FUNCTION "G7_STD_3" : VOID	// FC 72
AUTHOR : SIMATIC
FAMILY : S7GRAPH
NAME : SFMULTI
VERSION : 2.0
BEGIN
// (block stored without names or comments; labels and parameter names are numbered)
NETWORK
TITLE =
// (network holds code this reader does not know; not shown)
NETWORK
TITLE =
      L     DID [AR1,P#80.0];
      LAR2;
      L     DID [AR2,P#14.0];
      T     LD 30;
      L     DID [AR2,P#18.0];
      T     LD 40;
      L     DID [AR1,P#48.0];
      AD    DW#16#7FFFF;
      LAR2;
      AN    L 30.7;
      JC    M007;
      A     DIX [AR2,P#0.0];
      FP    DIX [AR1,P#7.4];
      S     DIX [AR1,P#11.4];
      +AR2  P#0.1;
M007: AN    L 30.6;
      JC    M008;
      A     DIX [AR2,P#0.0];
      FP    DIX [AR1,P#7.5];
      S     DIX [AR1,P#11.5];
      +AR2  P#0.1;
M008: AN    L 30.5;
      JC    M009;
      A     DIX [AR2,P#0.0];
      FP    DIX [AR1,P#9.3];
      S     DIX [AR1,P#13.3];
      +AR2  P#0.1;
M009: AN    L 30.4;
      JC    M010;
      A     DIX [AR2,P#0.0];
      FP    DIX [AR1,P#9.2];
      S     DIX [AR1,P#13.2];
      +AR2  P#0.1;
M010: AN    L 30.3;
      JC    M011;
      A     DIX [AR2,P#0.0];
      FP    DIX [AR1,P#6.4];
      S     DIX [AR1,P#10.4];
      +AR2  P#0.1;
M011: AN    L 30.2;
      JC    M012;
      A     DIX [AR2,P#0.0];
      FP    DIX [AR1,P#6.5];
      S     DIX [AR1,P#10.5];
      +AR2  P#0.1;
M012: AN    L 30.1;
      JC    M013;
      A     DIX [AR2,P#0.0];
      FP    DIX [AR1,P#7.6];
      X     DIX [AR1,P#11.6];
      =     DIX [AR1,P#11.6];
      +AR2  P#0.1;
M013: AN    L 30.0;
      JC    M014;
      A     DIX [AR2,P#0.0];
      FP    DIX [AR1,P#7.7];
      X     DIX [AR1,P#11.7];
      =     DIX [AR1,P#11.7];
      +AR2  P#0.1;
M014: AN    L 31.7;
      JC    M015;
      A     DIX [AR2,P#0.0];
      FP    DIX [AR1,P#8.0];
      X     DIX [AR1,P#12.0];
      =     DIX [AR1,P#12.0];
      +AR2  P#0.1;
M015: AN    L 31.6;
      JC    M016;
      A     DIX [AR2,P#0.0];
      FP    DIX [AR1,P#7.0];
      X     DIX [AR1,P#11.0];
      =     DIX [AR1,P#11.0];
      +AR2  P#0.1;
M016: AN    L 31.5;
      JC    M017;
      A     DIX [AR2,P#0.0];
      FP    DIX [AR1,P#7.1];
      X     DIX [AR1,P#11.1];
      =     DIX [AR1,P#11.1];
      +AR2  P#0.1;
M017: AN    L 31.4;
      JC    M018;
      A     DIX [AR2,P#0.0];
      FP    DIX [AR1,P#7.2];
      X     DIX [AR1,P#11.2];
      =     DIX [AR1,P#11.2];
      +AR2  P#0.1;
M018: AN    L 31.3;
      JC    M019;
      A     DIX [AR2,P#0.0];
      FP    DIX [AR1,P#7.3];
      X     DIX [AR1,P#11.3];
      =     DIX [AR1,P#11.3];
      +AR2  P#0.1;
M019: AN    L 31.2;
      JC    M020;
      A     DIX [AR2,P#0.0];
      FP    DIX [AR1,P#8.1];
      S     DIX [AR1,P#12.1];
      R     DIX [AR1,P#12.2];
      R     DIX [AR1,P#12.3];
      R     DIX [AR1,P#12.4];
      R     DIX [AR1,P#12.5];
      +AR2  P#0.1;
M020: AN    L 31.1;
      JC    M021;
      A     DIX [AR2,P#0.0];
      FP    DIX [AR1,P#8.2];
      R     DIX [AR1,P#12.1];
      S     DIX [AR1,P#12.2];
      R     DIX [AR1,P#12.3];
      R     DIX [AR1,P#12.4];
      R     DIX [AR1,P#12.5];
      +AR2  P#0.1;
M021: AN    L 31.0;
      JC    M022;
      A     DIX [AR2,P#0.0];
      FP    DIX [AR1,P#8.3];
      R     DIX [AR1,P#12.1];
      R     DIX [AR1,P#12.2];
      S     DIX [AR1,P#12.3];
      R     DIX [AR1,P#12.4];
      R     DIX [AR1,P#12.5];
      +AR2  P#0.1;
M022: AN    L 32.7;
      JC    M023;
      A     DIX [AR2,P#0.0];
      FP    DIX [AR1,P#8.4];
      S     DIX [AR1,P#12.4];
      +AR2  P#0.1;
M023: AN    L 32.6;
      JC    M024;
      A     DIX [AR2,P#0.0];
      FP    DIX [AR1,P#8.5];
      S     DIX [AR1,P#12.5];
      +AR2  P#0.1;
M024: AN    L 32.5;
      JC    M025;
      A     DIX [AR2,P#0.0];
      FP    DIX [AR1,P#6.0];
      =     L 29.1;
      S     DIX [AR1,P#10.0];
      R     DIX [AR1,P#10.2];
      R     DIX [AR1,P#10.3];
      R     DIX [AR1,P#10.1];
      +AR2  P#0.1;
      R     DIX [AR1,P#12.4];
      R     DIX [AR1,P#12.5];
      R     DIX [AR1,P#10.6];
      R     DIX [AR1,P#10.7];
      AN    L 31.2;
      AN    L 31.1;
      AN    L 31.0;
      A     L 29.1;
      S     DIX [AR1,P#12.1];
      R     DIX [AR1,P#12.2];
      R     DIX [AR1,P#12.3];
M025: AN    L 32.4;
      JC    M026;
      A     DIX [AR2,P#0.0];
      FP    DIX [AR1,P#6.2];
      =     L 29.1;
      R     DIX [AR1,P#10.0];
      S     DIX [AR1,P#10.2];
      R     DIX [AR1,P#10.3];
      R     DIX [AR1,P#10.1];
      +AR2  P#0.1;
      R     DIX [AR1,P#12.4];
      R     DIX [AR1,P#12.5];
      R     DIX [AR1,P#10.6];
      R     DIX [AR1,P#10.7];
      AN    L 31.2;
      AN    L 31.1;
      AN    L 31.0;
      A     L 29.1;
      S     DIX [AR1,P#12.1];
      R     DIX [AR1,P#12.2];
      R     DIX [AR1,P#12.3];
M026: AN    L 32.3;
      JC    M027;
      A     DIX [AR2,P#0.0];
      FP    DIX [AR1,P#6.3];
      =     L 29.1;
      R     DIX [AR1,P#10.0];
      R     DIX [AR1,P#10.2];
      S     DIX [AR1,P#10.3];
      R     DIX [AR1,P#10.1];
      +AR2  P#0.1;
      R     DIX [AR1,P#12.4];
      R     DIX [AR1,P#12.5];
      R     DIX [AR1,P#10.6];
      R     DIX [AR1,P#10.7];
      AN    L 31.2;
      AN    L 31.1;
      AN    L 31.0;
      A     L 29.1;
      S     DIX [AR1,P#12.1];
      R     DIX [AR1,P#12.2];
      R     DIX [AR1,P#12.3];
M027: AN    L 32.2;
      JC    M028;
      A     DIX [AR2,P#0.0];
      FP    DIX [AR1,P#6.1];
      =     L 29.1;
      R     DIX [AR1,P#10.0];
      R     DIX [AR1,P#10.2];
      R     DIX [AR1,P#10.3];
      S     DIX [AR1,P#10.1];
      +AR2  P#0.1;
      R     DIX [AR1,P#12.4];
      R     DIX [AR1,P#12.5];
      R     DIX [AR1,P#10.6];
      R     DIX [AR1,P#10.7];
      AN    L 31.2;
      AN    L 31.1;
      AN    L 31.0;
      A     L 29.1;
      R     DIX [AR1,P#12.1];
      R     DIX [AR1,P#12.2];
      S     DIX [AR1,P#12.3];
M028: AN    L 32.1;
      JC    M031;
      +AR2  P#1.7;
      TAR2;
      SRD   4;
      SLD   4;
      LAR2;
      AN    L 32.0;
      JC    M029;
      L     DIW [AR2,P#0.0];
      T     DIW [AR1,P#2.0];
      JU    M030;
M029: L     DIW [AR1,P#2.0];
      L     DIW [AR2,P#0.0];
      T     DIW [AR1,P#2.0];
      <>I;
      S     DIX [AR1,P#12.6];
M030: +AR2  P#2.0;
M031: AN    L 32.0;
      JC    M032;
      A     DIX [AR2,P#0.0];
      FP    DIX [AR1,P#8.6];
      S     DIX [AR1,P#12.6];
      +AR2  P#0.1;
M032: AN    L 33.7;
      JC    M033;
      A     DIX [AR2,P#0.0];
      FP    DIX [AR1,P#8.7];
      S     DIX [AR1,P#12.7];
      +AR2  P#0.1;
M033: AN    L 33.6;
      JC    M034;
      A     DIX [AR2,P#0.0];
      FP    DIX [AR1,P#9.0];
      S     DIX [AR1,P#13.0];
      +AR2  P#0.1;
M034: AN    L 33.5;
      JC    M035;
      A     DIX [AR2,P#0.0];
      FP    DIX [AR1,P#6.6];
      S     DIX [AR1,P#10.6];
      +AR2  P#0.1;
M035: AN    L 33.4;
      JC    M036;
      A     DIX [AR2,P#0.0];
      FP    DIX [AR1,P#6.7];
      S     DIX [AR1,P#10.7];
      +AR2  P#0.1;
M036: AN    L 33.3;
      JC    M037;
      A     DIX [AR2,P#0.0];
      FP    DIX [AR1,P#9.1];
      S     DIX [AR1,P#13.1];
M037: NOP   0;
NETWORK
TITLE =
      BLD   7;
      UC    "TIME_TCK";
      {     P#L 8.0 };
      BLD   8;
      L     LD 8;
      T     DID [AR1,P#22.0];
      A     DIX [AR1,P#11.7];
      JC    M038;
      L     DID [AR1,P#18.0];
      -D;
      T     DID [AR1,P#14.0];
      AD    DW#16#FFFFF000;
      JZ    M039;
M038: L     B#16#0;
      T     DID [AR1,P#14.0];
M039: L     DID [AR1,P#22.0];
      T     DID [AR1,P#18.0];
NETWORK
TITLE =
      L     DID [AR1,P#48.0];
      LAR2;
      L     DIW [AR1,P#52.0];
      T     LW 12;
      SET;
      S     DIX [AR1,P#27.5];
      AN    DIX [AR1,P#13.6];
      JC    M040;
      A     DIX [AR1,P#10.1];
      =     DIX [AR1,P#13.4];
M040: LAR1  LD 0;
      L     B#16#1;
      T     DIB [AR1,P#30.0];
      UC    FB [LW 12];
NETWORK
TITLE =
      LAR1  LD 4;
      L     DID [AR1,P#14.0];
      T     LW 22;
      CLR;
      LAR1  LD 0;
      L     DID [AR1,P#4.0];
      T     LD 8;
      LAR1;
      L     DIB [AR1,P#0.0];
      JU    M045;
M041: T     LB 16;
      +AR1  P#1.0;
      L     DIB [AR1,P#0.0];
      SLW   7;
      LAR2  LD 0;
      +AR2;
      +AR2;
      L     DID [AR2,P#4.0];
      L     LW 22;
      +D;
      <=D;
      JC    M042;
      L     DW#16#7FFFFFFF;
M042: T     DID [AR2,P#4.0];
      O     DIX [AR2,P#1.1];
      O     DIX [AR2,P#1.2];
      JC    M044;
      L     DID [AR2,P#8.0];
      L     LW 22;
      +D;
      <=D;
      JC    M043;
      L     DW#16#7FFFFFFF;
M043: T     DID [AR2,P#8.0];
M044: L     LB 16;
M045: LOOP  M041;
NETWORK
TITLE =
      LAR1  LD 4;
      L     DID [AR1,P#40.0];
      LAR1;
      SET;
      R     L 29.0;
      JU    M285;
M046: LAR1  LD 8;
      SET;
      S     L 29.0;
      JU    M285;
M047: LAR1  LD 4;
      L     DID [AR1,P#44.0];
      LAR2;
      L     B#16#1;
      T     DIB [AR2,P#0.0];
      L     DID [AR1,P#40.0];
      LAR2;
      L     B#16#1;
      T     DIB [AR2,P#0.0];
      L     DID [AR1,P#36.0];
      LAR2;
      L     B#16#1;
      T     DIB [AR2,P#0.0];
      LAR1  LD 8;
      L     B#16#0;
      JU    M251;
M048: NOP   0;
NETWORK
TITLE =
      LAR1  LD 4;
      AN    DIX [AR1,P#11.4];
      JC    M050;
      R     DIX [AR1,P#11.4];
      R     DIX [AR1,P#11.5];
      LAR1  LD 8;
      L     B#16#0;
      JU    M261;
M049: JU    M080;
M050: NOP   0;
NETWORK
TITLE =
      LAR1  LD 4;
      AN    DIX [AR1,P#11.5];
      JC    M056;
      R     DIX [AR1,P#11.5];
      R     DIX [AR1,P#26.4];
      R     DIX [AR1,P#26.5];
      R     DIX [AR1,P#26.6];
      R     DIX [AR1,P#26.7];
      R     DIX [AR1,P#27.0];
      R     DIX [AR1,P#26.3];
      LAR1  LD 8;
      L     B#16#1;
      JU    M261;
M051: LAR1  LD 0;
      L     DIW [AR1,P#28.0];
      SLD   3;
      LAR1;
      L     B#16#0;
      JU    M256;
M052: LAR1  LD 4;
      L     DID [AR1,P#40.0];
      LAR1;
      L     B#16#4;
      JU    M270;
M053: LAR1  LD 4;
      L     DID [AR1,P#36.0];
      T     LD 8;
      LAR1;
      L     B#16#3;
      JU    M270;
M054: LAR1  LD 8;
      L     B#16#1;
      JU    M251;
M055: JU    M080;
M056: NOP   0;
NETWORK
TITLE =
      LAR1  LD 4;
      AN    DIX [AR1,P#13.3];
      AN    DIX [AR1,P#13.2];
      JC    M060;
      A     DIX [AR1,P#13.3];
      R     DIX [AR1,P#26.1];
      R     DIX [AR1,P#26.2];
      R     DIX [AR1,P#26.0];
      R     DIX [AR1,P#26.4];
      R     DIX [AR1,P#26.5];
      R     DIX [AR1,P#26.6];
      R     DIX [AR1,P#26.7];
      R     DIX [AR1,P#27.0];
      R     DIX [AR1,P#26.3];
      LAR2  LD 0;
      L     DIW [AR2,P#18.0];
      SLD   3;
      T     LD 24;
      L     DIB [LD 24];
      JU    M059;
M057: T     LB 17;
      L     LD 24;
      +     L#8;
      T     LD 24;
      L     DIB [LD 24];
      SLW   7;
      LAR2  LD 0;
      +AR2;
      +AR2;
      A     DIX [AR1,P#13.2];
      S     DIX [AR2,P#0.3];
      AN    DIX [AR1,P#13.3];
      JC    M058;
      S     DIX [AR2,P#0.4];
      R     DIX [AR2,P#1.2];
      L     B#16#0;
      T     DID [AR2,P#8.0];
M058: L     LB 17;
M059: LOOP  M057;
      R     DIX [AR1,P#13.2];
M060: R     DIX [AR1,P#13.3];
NETWORK
TITLE =
      AN    DIX [AR1,P#10.4];
      AN    DIX [AR1,P#10.5];
      JC    M061;
      L     B#16#0;
      L     DIB [AR1,P#4.0];
      ==I;
      JC    M061;
      SLW   7;
      LAR2  LD 0;
      +AR2;
      +AR2;
      A     DIX [AR1,P#10.5];
      A(;
      O     DIX [AR2,P#1.1];
      O     DIX [AR2,P#1.2];
      );
      S     DIX [AR2,P#0.3];
      A     DIX [AR1,P#10.4];
      A(;
      O     DIX [AR2,P#1.1];
      O     DIX [AR2,P#1.2];
      );
      JCN   M061;
      S     DIX [AR2,P#0.4];
      R     DIX [AR2,P#1.2];
      L     B#16#0;
      T     DID [AR2,P#8.0];
M061: R     DIX [AR1,P#10.5];
      R     DIX [AR1,P#10.4];
NETWORK
TITLE =
      AN    DIX [AR1,P#12.4];
      JC    M064;
      L     B#16#0;
      L     DIB [AR1,P#4.0];
      ==I;
      JC    M064;
      L     B#16#2;
      L     DIB [AR1,P#4.0];
      >I;
      JC    M062;
      DEC   1;
      JU    M063;
M062: L     DID [AR1,P#80.0];
      LAR2;
      L     DIB [AR2,P#12.0];
M063: T     DIB [AR1,P#4.0];
      A     DIX [AR1,P#12.3];
      JC    M064;
      SLW   7;
      LAR2  LD 0;
      +AR2;
      +AR2;
      A     DIX [AR1,P#12.1];
      A     DIX [AR2,P#1.0];
      O;
      A     DIX [AR1,P#12.2];
      A(;
      O     DIX [AR2,P#1.1];
      O     DIX [AR2,P#1.2];
      );
M064: R     DIX [AR1,P#12.4];
NETWORK
TITLE =
      AN    DIX [AR1,P#12.5];
      JC    M066;
      L     B#16#0;
      L     DIB [AR1,P#4.0];
      ==I;
      JC    M066;
      L     DID [AR1,P#80.0];
      LAR2;
      L     DIB [AR2,P#12.0];
      L     DIB [AR1,P#4.0];
      INC   1;
      >=I;
      JC    M065;
      L     B#16#1;
M065: T     DIB [AR1,P#4.0];
      A     DIX [AR1,P#12.3];
      JC    M066;
      SLW   7;
      LAR2  LD 0;
      +AR2;
      +AR2;
      A     DIX [AR1,P#12.1];
      A     DIX [AR2,P#1.0];
      O;
      A     DIX [AR1,P#12.2];
      A(;
      O     DIX [AR2,P#1.1];
      O     DIX [AR2,P#1.2];
      );
M066: R     DIX [AR1,P#12.5];
NETWORK
TITLE =
      ON    DIX [AR1,P#10.1];
      ON    DIX [AR1,P#12.6];
      JC    M068;
      L     DIW [AR1,P#2.0];
      L     B#16#2;
      JU    M266;
M067: TAK;
      L     B#16#0;
      ==I;
      JC    M068;
      TAK;
      T     DIB [AR1,P#4.0];
M068: R     DIX [AR1,P#12.6];
NETWORK
TITLE =
      AN    DIX [AR1,P#10.1];
      R     DIX [AR1,P#12.7];
      AN    DIX [AR1,P#12.7];
      JC    M070;
      R     DIX [AR1,P#12.7];
      L     DIW [AR1,P#0.0];
      L     B#16#0;
      JU    M266;
M069: <>I;
      R     L 29.0;
      TAK;
      JC    M288;
M070: LAR1  LD 4;
      L     DID [AR1,P#68.0];
      T     LD 8;
      LAR1;
      LAR2  LD 0;
      L     DIB [AR2,P#26.0];
      SLW   3;
      +AR1;
      L     B#16#1;
      JU    M256;
M071: NOP   0;
NETWORK
TITLE =
      LAR1  LD 4;
      AN    DIX [AR1,P#10.1];
      R     DIX [AR1,P#13.0];
      AN    DIX [AR1,P#13.0];
      JC    M073;
      R     DIX [AR1,P#13.0];
      LAR2  LD 0;
      L     DID [AR2,P#4.0];
      LAR2;
      L     DIB [AR2,P#0.0];
      L     B#16#1;
      ==I;
      S     DIX [AR1,P#26.5];
      JC    M073;
      L     DIW [AR1,P#0.0];
      L     B#16#1;
      JU    M266;
M072: TAK;
      L     B#16#0;
      <>I;
      S     L 29.0;
      TAK;
      JC    M288;
M073: LAR1  LD 8;
      L     B#16#2;
      JU    M261;
M074: NOP   0;
NETWORK
TITLE =
      LAR1  LD 4;
      AN    DIX [AR1,P#10.6];
      JC    M077;
      L     B#16#0;
      L     DIB [AR1,P#5.0];
      ==I;
      JC    M077;
      L     B#16#2;
      L     DIB [AR1,P#5.0];
      >I;
      JC    M075;
      DEC   1;
      JU    M076;
M075: L     DID [AR1,P#80.0];
      LAR2;
      L     DIB [AR2,P#9.0];
M076: T     DIB [AR1,P#5.0];
      LAR2  LD 0;
      L     DIW [AR2,P#12.0];
      SLD   3;
      LAR2;
      TAK;
      SLW   7;
      +AR2;
      O(;
      O     DIX [AR1,P#10.0];
      O     DIX [AR1,P#10.3];
      A     DIX [AR2,P#0.0];
      );
      O(;
      O     DIX [AR1,P#10.1];
      O     DIX [AR1,P#10.2];
      A     DIX [AR2,P#0.1];
      );
M077: R     DIX [AR1,P#10.6];
NETWORK
TITLE =
      AN    DIX [AR1,P#10.7];
      JC    M079;
      L     B#16#0;
      L     DIB [AR1,P#5.0];
      ==I;
      JC    M079;
      L     DID [AR1,P#80.0];
      LAR2;
      L     DIB [AR2,P#9.0];
      L     DIB [AR1,P#5.0];
      INC   1;
      >=I;
      JC    M078;
      L     B#16#1;
M078: T     DIB [AR1,P#5.0];
      LAR2  LD 0;
      L     DIW [AR2,P#12.0];
      SLD   3;
      LAR2;
      TAK;
      SLW   7;
      +AR2;
      O(;
      O     DIX [AR1,P#10.0];
      O     DIX [AR1,P#10.3];
      A     DIX [AR2,P#0.0];
      );
      O(;
      O     DIX [AR1,P#10.1];
      O     DIX [AR1,P#10.2];
      A     DIX [AR2,P#0.1];
      );
M079: R     DIX [AR1,P#10.7];
NETWORK
TITLE =
M080: LAR1  LD 4;
      L     DID [AR1,P#68.0];
      LAR1;
      L     B#16#1;
      T     DIB [AR1,P#0.0];
      LAR2  LD 0;
      L     DIB [AR2,P#26.0];
      SLW   3;
      +AR1;
      TAK;
      T     DIB [AR1,P#0.0];
NETWORK
TITLE =
M081: SET;
      LAR1  LD 0;
      L     DIW [AR1,P#12.0];
      SLD   3;
      T     LD 8;
      L     DIW [AR1,P#14.0];
      SLD   3;
      LAR1;
      L     DIB [AR1,P#0.0];
      JU    M083;
M082: +AR1  P#1.0;
      L     DIB [AR1,P#0.0];
      SLW   7;
      LAR2  LD 8;
      +AR2;
      R     DIX [AR2,P#0.0];
      R     DIX [AR2,P#0.1];
      R     DIX [AR2,P#0.2];
      TAK;
M083: LOOP  M082;
      LAR1  LD 0;
      L     DIW [AR1,P#14.0];
      SLD   3;
      LAR2;
      L     B#16#1;
      T     DIB [AR2,P#0.0];
      L     DIB [AR1,P#25.0];
      SLW   3;
      +AR2;
      L     B#16#1;
      T     DIB [AR2,P#0.0];
      TAK;
      +AR2;
      L     B#16#1;
      T     DIB [AR2,P#0.0];
NETWORK
TITLE =
      LAR1  LD 4;
      L     DID [AR1,P#44.0];
      T     LD 8;
      L     DID [AR1,P#80.0];
      LAR2;
      L     DIB [AR2,P#6.0];
      T     LW 22;
      LAR2  LD 0;
      L     DIW [AR2,P#20.0];
      L     DIB [AR2,P#2.0];
      SLW   1;
      +D;
      SLD   3;
      T     LD 24;
      L     DIW [AR2,P#22.0];
      SLD   3;
      T     LD 4;
      L     DIB [LD 8];
      JU    M093;
M084: T     LB 17;
      L     LD 8;
      +     L#8;
      T     LD 8;
      L     DIB [LD 8];
      T     LB 14;
M085: SLW   7;
      LAR1  AR2;
      +AR1;
      +AR1;
      ON    DIX [AR1,P#24.0];
      O     DIX [AR1,P#0.5];
      JC    M092;
      LAR1  LD 4;
      SRW   4;
      +AR1;
      L     LB 14;
      L     DIB [AR1,P#0.0];
      <>I;
      JC    M085;
      LAR1  LD 4;
      SLW   3;
      +AR1;
      L     DIB [AR2,P#3.0];
      SLW   3;
      +AR1;
      +AR1;
      +AR1;
      L     DIB [AR1,P#0.0];
      T     LB 16;
      L     DIW [AR2,P#12.0];
      SLD   3;
      LAR1;
      TAK;
      SLW   7;
      +AR1;
      A     DIX [AR1,P#0.0];
      JC    M092;
      SRW   7;
M086: T     LB 15;
      L     DIW [AR2,P#20.0];
      SLD   3;
      LAR1;
      TAK;
      SLW   3;
      +AR1;
      L     DIB [AR1,P#0.0];
      L     DIB [AR2,P#2.0];
      SLW   5;
      +AR1;
      TAK;
      L     DIB [AR1,P#0.0];
      <>I;
      JC    M087;
      SLW   7;
      LAR1  AR2;
      +AR1;
      +AR1;
      A     DIX [AR1,P#24.0];
      JC    M092;
      JU    M089;
M087: T     LB 14;
M088: SLW   7;
      LAR1  AR2;
      +AR1;
      +AR1;
      A     DIX [AR1,P#24.0];
      JC    M092;
      L     DIB [AR2,P#3.0];
      SLW   3;
      LAR1  LD 4;
      +AR1;
      TAK;
      SRW   4;
      +AR1;
      L     LB 14;
      L     DIB [AR1,P#0.0];
      <>I;
      JC    M088;
M089: LAR1  LD 24;
      L     LB 15;
      SLW   3;
      +AR1;
      L     LB 16;
      L     DIB [AR1,P#0.0];
      <>I;
      JC    M086;
M090: T     LB 15;
      L     DIW [AR2,P#14.0];
      SLD   3;
      LAR1;
      L     LW 22;
      L     DIB [AR1,P#0.0];
      >=I;
      JC    M091;
      L     DID [AR2,P#8.0];
      LAR1;
      S     DIX [AR1,P#26.7];
      JU    M094;
M091: INC   1;
      T     DIB [AR1,P#0.0];
      DEC   1;
      SLW   3;
      +AR1;
      L     LB 15;
      T     DIB [AR1,P#0.0];
      L     DIW [AR2,P#12.0];
      SLD   3;
      LAR1;
      TAK;
      SLW   7;
      +AR1;
      S     DIX [AR1,P#0.0];
      LAR1  LD 24;
      SRW   4;
      +AR1;
      L     LB 16;
      L     DIB [AR1,P#0.0];
      <>I;
      JC    M090;
M092: L     LB 17;
M093: LOOP  M084;
M094: L     DID [AR2,P#8.0];
      T     LD 4;
NETWORK
TITLE =
      LAR1  LD 4;
      CLR;
      A     DIX [AR1,P#13.5];
      =     L 29.7;
      O     DIX [AR1,P#10.6];
      O     DIX [AR1,P#10.7];
      A     L 41.6;
      R     DIX [AR1,P#13.1];
      L     DIW [AR2,P#14.0];
      SLD   3;
      T     LD 8;
      LAR1;
      L     DIB [AR2,P#25.0];
      SLW   3;
      T     LW 22;
      +D;
      T     LD 24;
      L     DIB [AR1,P#0.0];
      T     LB 16;
      SLW   3;
      +AR1;
      L     B#16#0;
      T     DIB [AR1,P#0.0];
      T     LB 15;
      AN    L 29.7;
      JC    M095;
      LAR1  LD 4;
      L     DID [AR1,P#80.0];
      LAR1;
      L     DIB [AR1,P#9.0];
      INC   1;
      T     LB 16;
M095: L     LB 16;
      JU    M101;
M096: T     LB 16;
      LAR1  LD 4;
      L     B#16#0;
      T     DID [AR1,P#72.0];
      L     DID [AR1,P#48.0];
      LAR2;
      A     L 29.7;
      JC    M097;
      L     LD 8;
      +     L#8;
      T     LD 8;
      L     DIB [LD 8];
      JU    M098;
M097: L     LB 15;
      INC   1;
M098: T     LB 15;
      LAR1  LD 0;
      T     DIB [AR1,P#31.0];
      L     B#16#2;
      T     DIB [AR1,P#30.0];
      UC    FB [LW 12];
      LAR1  LD 0;
      L     DIW [AR1,P#12.0];
      SLD   3;
      LAR1;
      L     LB 15;
      SLW   7;
      +AR1;
      =     DIX [AR1,P#0.1];
      LAR2  LD 4;
      AN    DIX [AR1,P#0.0];
      JC    M099;
      O(;
      SRW   7;
      L     DIB [AR2,P#5.0];
      ==I;
      A     L 41.6;
      A     DIX [AR2,P#10.3];
      A     DIX [AR2,P#13.1];
      );
      O(;
      AN    L 41.6;
      A     DIX [AR2,P#10.3];
      A     DIX [AR2,P#13.1];
      );
      R     DIX [AR2,P#13.1];
      S     DIX [AR1,P#0.1];
      L     DID [AR1,P#4.0];
      T     DID [AR1,P#8.0];
M099: L     DID [AR2,P#72.0];
      T     DID [AR1,P#4.0];
      ON    DIX [AR1,P#0.0];
      ON    DIX [AR1,P#0.1];
      JC    M100;
      LAR1  LD 24;
      L     DIB [AR1,P#0.0];
      INC   1;
      T     DIB [AR1,P#0.0];
      DEC   1;
      SLW   3;
      +AR1;
      L     LB 15;
      T     DIB [AR1,P#0.0];
M100: L     LB 16;
M101: LOOP  M096;
NETWORK
TITLE =
// (network holds code this reader does not know; not shown)
NETWORK
TITLE =
// (network holds code this reader does not know; not shown)
NETWORK
TITLE =
      LAR1  LD 0;
      L     DIB [AR1,P#2.0];
      SLW   3;
      L     LD 24;
      +D;
      T     LD 24;
      L     DID [AR1,P#8.0];
      LAR1;
      L     DID [AR1,P#36.0];
      T     LD 4;
      LAR2  LD 8;
      L     DIB [AR2,P#0.0];
      JU    M117;
M113: T     LB 17;
      +AR2  P#1.0;
      LAR1  LD 24;
      L     DIB [AR2,P#0.0];
      T     LB 15;
      SLW   3;
      +AR1;
      L     B#16#0;
      L     DIB [AR1,P#0.0];
      ==I;
      JC    M116;
      T     LB 14;
M114: T     LB 16;
      SLW   7;
      LAR1  LD 0;
      +AR1;
      +AR1;
      O     DIX [AR1,P#0.0];
      O     DIX [AR1,P#1.0];
      JC    M115;
      S     DIX [AR1,P#0.0];
      S     DIX [AR1,P#1.0];
      LAR1  LD 4;
      L     DIB [AR1,P#0.0];
      INC   1;
      T     DIB [AR1,P#0.0];
      DEC   1;
      SLW   3;
      +AR1;
      L     LB 16;
      T     DIB [AR1,P#0.0];
      LAR1  LD 0;
      L     DIW [AR1,P#20.0];
      SLD   3;
      LAR1;
      L     LB 15;
      SLW   3;
      +AR1;
      L     DIB [AR1,P#0.0];
      L     B#16#0;
      <>I;
      JC    M116;
M115: LAR1  LD 0;
      L     DIW [AR1,P#22.0];
      L     DIB [AR1,P#3.0];
      +D;
      SLD   3;
      LAR1;
      L     LB 16;
      SLW   3;
      +AR1;
      L     LB 14;
      L     DIB [AR1,P#0.0];
      <>I;
      JC    M114;
M116: L     LB 17;
M117: LOOP  M113;
NETWORK
TITLE =
      LAR1  LD 4;
      LAR2  LD 0;
      L     DID [AR2,P#8.0];
      T     LD 4;
      L     B#16#2;
      JU    M251;
M118: NOP   0;
NETWORK
TITLE =
      LAR1  LD 8;
      LAR2  LD 4;
      L     B#16#1;
      L     DIB [AR1,P#0.0];
      <I;
      A     DIX [AR2,P#11.3];
      JC    M081;
NETWORK
TITLE =
      L     DID [AR2,P#44.0];
      LAR1;
      L     DIB [AR1,P#0.0];
      JU    M120;
M119: +AR1  P#1.0;
      L     DIB [AR1,P#0.0];
      SLW   7;
      LAR2  LD 0;
      +AR2;
      +AR2;
      R     DIX [AR2,P#24.0];
      TAK;
M120: LOOP  M119;
NETWORK
TITLE =
      LAR1  LD 4;
      L     DID [AR1,P#80.0];
      LAR2;
      AN    DIX [AR2,P#34.7];
      JC    M129;
      L     DIW [AR2,P#32.0];
      T     LW 18;
      L     B#16#2;
      -D;
      SLD   3;
      LAR2;
      L     DIW [AR2,P#0.0];
      T     LW 20;
      L     LW 18;
      LAR2  LD 0;
      L     DIB [AR2,P#3.0];
      INC   2;
      -D;
      SLD   3;
      T     LD 8;
      L     DIB [LD 8];
      T     LW 18;
      L     DID [AR1,P#36.0];
      T     LD 24;
      L     DIB [LD 24];
      JU    M128;
M121: T     LB 17;
      L     LD 24;
      +     L#8;
      T     LD 24;
      L     DIB [LD 24];
      SLW   3;
      LAR1  LD 8;
      +AR1;
      L     DIB [AR1,P#0.0];
      T     LW 22;
      SET;
      =     L 29.6;
      LAR1  LD 0;
      L     DID [AR1,P#4.0];
      LAR2;
M122: L     DIB [AR2,P#0.0];
      JU    M126;
M123: T     LB 14;
      +AR2  P#1.0;
      L     DIB [LD 24];
      L     DIB [AR2,P#0.0];
      <>I;
      JC    M124;
      A     L 29.6;
      JC    M125;
      L     B#16#1;
      T     LB 14;
      JC    M125;
M124: T     LB 16;
      SLW   3;
      LAR1  LD 8;
      +AR1;
      L     DIB [AR1,P#0.0];
      L     LW 18;
      *D;
      L     LW 22;
      +D;
      L     LW 20;
      SLD   3;
      +D;
      LAR1;
      A     DIX [AR1,P#0.0];
      JC    M125;
      L     LB 16;
      SLW   7;
      LAR1  LD 0;
      +AR1;
      +AR1;
      O     DIX [AR1,P#0.5];
      ON    DIX [AR1,P#1.0];
      JC    M125;
      S     DIX [AR1,P#0.5];
      R     DIX [AR1,P#1.0];
      LAR1  LD 4;
      L     DID [AR1,P#40.0];
      LAR1;
      L     DIB [AR1,P#0.0];
      INC   1;
      T     DIB [AR1,P#0.0];
      DEC   1;
      SLW   3;
      +AR1;
      L     LB 16;
      T     DIB [AR1,P#0.0];
M125: L     LB 14;
M126: LOOP  M123;
      AN    L 29.6;
      JC    M127;
      R     L 29.6;
      LAR1  LD 4;
      L     DID [AR1,P#36.0];
      LAR2;
      JU    M122;
M127: L     LB 17;
M128: LOOP  M121;
M129: NOP   0;
NETWORK
TITLE =
      LAR1  LD 4;
      L     DID [AR1,P#40.0];
      LAR1;
      L     B#16#2;
      JU    M270;
M130: NOP   0;
NETWORK
TITLE =
      LAR1  LD 4;
      L     DID [AR1,P#36.0];
      T     LD 8;
      LAR1;
      L     B#16#1;
      JU    M270;
M131: NOP   0;
NETWORK
TITLE =
      LAR1  LD 8;
      L     DIB [AR1,P#0.0];
      JU    M133;
M132: T     LB 14;
      +AR1  P#1.0;
      L     DIB [AR1,P#0.0];
      SLW   7;
      LAR2  LD 0;
      +AR2;
      +AR2;
      L     B#16#0;
      T     DID [AR2,P#4.0];
      T     DID [AR2,P#8.0];
      L     LB 14;
M133: LOOP  M132;
NETWORK
TITLE =
      LAR1  LD 0;
      L     DID [AR1,P#4.0];
      T     LD 8;
      LAR2;
      LAR1  LD 4;
      L     DID [AR1,P#44.0];
      LAR1;
      L     DIB [AR2,P#0.0];
M134: L     DIB [AR2,P#0.0];
      T     DIB [AR1,P#0.0];
      +AR1  P#1.0;
      +AR2  P#1.0;
      TAK;
      LOOP  M134;
      LAR1  LD 4;
      SET;
      S     DIX [AR1,P#27.6];
      LAR1  LD 8;
      L     B#16#0;
      JU    M270;
M135: NOP   0;
NETWORK
TITLE =
      LAR1  LD 4;
      L     DID [AR1,P#80.0];
      LAR2;
      L     DIB [AR2,P#7.0];
      T     LB 14;
      L     DID [AR1,P#36.0];
      LAR1;
      L     DIB [AR1,P#0.0];
      DEC   1;
      LAR2  LD 8;
      L     DIB [AR2,P#0.0];
      DEC   1;
      +I;
      L     LB 14;
      <=I;
      JC    M137;
      LAR2  LD 4;
      S     DIX [AR2,P#26.6];
      -I;
      T     LB 14;
      L     DIB [AR1,P#0.0];
      TAK;
      -I;
      T     DIB [AR1,P#0.0];
      SLW   3;
      +AR1;
      L     LB 14;
M136: T     LB 14;
      L     DIB [AR1,P#0.0];
      SLW   7;
      LAR2  LD 0;
      +AR2;
      +AR2;
      L     B#16#0;
      T     DIW [AR2,P#0.0];
      +AR1  P#1.0;
      L     LB 14;
      LOOP  M136;
M137: NOP   0;
NETWORK
TITLE =
// (network holds code this reader does not know; not shown)
NETWORK
TITLE =
      LAR1  LD 0;
      L     DIW [AR1,P#16.0];
      L     DIB [AR1,P#26.0];
      +D;
      SLD   3;
      LAR1;
      LAR2  LD 4;
      L     DID [AR2,P#40.0];
      LAR2;
      L     DIB [AR2,P#0.0];
M170: L     DIB [AR2,P#0.0];
      T     DIB [AR1,P#0.0];
      +AR1  P#1.0;
      +AR2  P#1.0;
      TAK;
      LOOP  M170;
      LAR1  LD 4;
      L     DID [AR1,P#36.0];
      LAR1;
      LAR2  LD 0;
      L     DID [AR2,P#4.0];
      LAR2;
      L     DIB [AR2,P#0.0];
      T     LB 14;
      L     DIB [AR1,P#0.0];
      DEC   1;
      +I;
      T     DIB [AR2,P#0.0];
      L     LB 14;
      SLW   3;
      +AR2;
      L     DIB [AR1,P#0.0];
      JU    M172;
M171: +AR1  P#1.0;
      L     DIB [AR1,P#0.0];
      T     DIB [AR2,P#0.0];
      +AR2  P#1.0;
      TAK;
M172: LOOP  M171;
      LAR1  LD 4;
      SET;
      R     DIX [AR1,P#27.6];
NETWORK
TITLE =
      LAR1  LD 0;
      L     B#16#6;
      T     DIB [AR1,P#30.0];
      LAR1  LD 4;
      L     DID [AR1,P#48.0];
      LAR2;
      UC    FB [LW 12];
      LAR1  LD 4;
      SET;
      R     DIX [AR1,P#27.5];
NETWORK
TITLE =
      LAR1  LD 0;
      L     DIW [AR1,P#18.0];
      SLD   3;
      T     LD 8;
      LAR1  LD 4;
      SET;
      R     DIX [AR1,P#26.1];
      R     DIX [AR1,P#26.2];
      L     DIB [LD 8];
      JU    M174;
M173: T     LB 14;
      L     LD 8;
      +     L#8;
      T     LD 8;
      L     DIB [LD 8];
      SLW   7;
      LAR2  LD 0;
      +AR2;
      +AR2;
      A     DIX [AR2,P#1.1];
      S     DIX [AR1,P#26.1];
      A     DIX [AR2,P#1.2];
      S     DIX [AR1,P#26.2];
      L     LB 14;
M174: LOOP  M173;
      O     DIX [AR1,P#26.1];
      O     DIX [AR1,P#26.2];
      =     DIX [AR1,P#26.0];
      O     DIX [AR1,P#26.4];
      O     DIX [AR1,P#26.5];
      O     DIX [AR1,P#26.6];
      O     DIX [AR1,P#26.7];
      O     DIX [AR1,P#27.0];
      =     DIX [AR1,P#26.3];
NETWORK
TITLE =
// (network holds code this reader does not know; not shown)
NETWORK
TITLE =
      CLR;
      AN    DIX [AR1,P#26.3];
      SAVE;
      L     DID [AR1,P#48.0];
      LAR2;
      BE;
NETWORK
TITLE =
M251: T     LB 28;
      LAR2  LD 4;
      L     DID [AR2,P#44.0];
      T     LD 24;
      CLR;
      L     DIB [AR1,P#0.0];
      JU    M254;
M252: T     LB 17;
      +AR1  P#1.0;
      L     DIB [AR1,P#0.0];
      SLW   7;
      LAR2  LD 0;
      +AR2;
      +AR2;
      A     DIX [AR2,P#24.0];
      JC    M253;
      S     DIX [AR2,P#24.0];
      LAR2  LD 24;
      L     DIB [AR2,P#0.0];
      INC   1;
      T     DIB [AR2,P#0.0];
      DEC   1;
      SLW   3;
      +AR2;
      TAK;
      SRW   7;
      T     DIB [AR2,P#0.0];
M253: L     LB 17;
M254: LOOP  M252;
      L     LB 28;
      JL    M255;
      JU    M048;
      JU    M055;
      JU    M118;
M255: NOP   0;
NETWORK
TITLE =
M256: T     LB 28;
      LAR2  LD 4;
      L     DID [AR2,P#36.0];
      T     LD 24;
      CLR;
      L     DIB [AR1,P#0.0];
      JU    M259;
M257: T     LB 17;
      +AR1  P#1.0;
      L     DIB [AR1,P#0.0];
      SLW   7;
      LAR2  LD 0;
      +AR2;
      +AR2;
      O     DIX [AR2,P#0.0];
      O     DIX [AR2,P#1.0];
      JC    M258;
      S     DIX [AR2,P#0.0];
      S     DIX [AR2,P#1.0];
      LAR2  LD 24;
      L     DIB [AR2,P#0.0];
      INC   1;
      T     DIB [AR2,P#0.0];
      DEC   1;
      SLW   3;
      +AR2;
      TAK;
      SRW   7;
      T     DIB [AR2,P#0.0];
M258: L     LB 17;
M259: LOOP  M257;
      L     LB 28;
      JL    M260;
      JU    M052;
      JU    M071;
M260: NOP   0;
NETWORK
TITLE =
M261: T     LB 28;
      LAR2  LD 4;
      L     DID [AR2,P#40.0];
      T     LD 24;
      CLR;
      L     DIB [AR1,P#0.0];
      JU    M264;
M262: T     LB 17;
      +AR1  P#1.0;
      L     DIB [AR1,P#0.0];
      SLW   7;
      LAR2  LD 0;
      +AR2;
      +AR2;
      O     DIX [AR2,P#0.5];
      ON    DIX [AR2,P#1.0];
      JC    M263;
      S     DIX [AR2,P#0.5];
      R     DIX [AR2,P#1.0];
      LAR2  LD 24;
      L     DIB [AR2,P#0.0];
      INC   1;
      T     DIB [AR2,P#0.0];
      DEC   1;
      SLW   3;
      +AR2;
      TAK;
      SRW   7;
      T     DIB [AR2,P#0.0];
M263: L     LB 17;
M264: LOOP  M262;
      L     LB 28;
      JL    M265;
      JU    M049;
      JU    M051;
      JU    M074;
M265: NOP   0;
NETWORK
TITLE =
M266: T     LB 28;
      TAK;
      T     LW 20;
      L     B#16#0;
      T     LW 18;
      L     DID [AR1,P#80.0];
      LAR2;
      L     DIB [AR2,P#12.0];
      LAR2  LD 0;
M267: T     LB 17;
      L     LW 18;
      INC   1;
      T     LW 18;
      +AR2  P#32.0;
      L     LW 20;
      L     DIW [AR2,P#2.0];
      ==I;
      L     LW 18;
      JC    M268;
      L     LB 17;
      LOOP  M267;
      S     DIX [AR1,P#26.4];
M268: L     LB 28;
      JL    M269;
      JU    M069;
      JU    M072;
      JU    M067;
M269: NOP   0;
NETWORK
TITLE =
M270: T     LB 28;
      CLR;
      TAR1  LD 24;
      L     DIB [AR1,P#0.0];
      L     B#16#1;
      T     DIB [AR1,P#0.0];
      TAK;
      JU    M278;
M271: T     LB 17;
      +AR1  P#1.0;
      L     DIB [AR1,P#0.0];
      SLW   7;
      LAR2  LD 0;
      +AR2;
      +AR2;
      L     LB 28;
      JL    M272;
      JU    M273;
      JU    M275;
      JU    M274;
      JU    M275;
      JU    M274;
M272: NOP   0;
M273: A     DIX [AR2,P#0.5];
      JC    M277;
      JU    M276;
M274: A     DIX [AR2,P#0.5];
      A     DIX [AR2,P#0.0];
      R     DIX [AR2,P#0.5];
      R     DIX [AR2,P#0.0];
      JC    M277;
      JU    M276;
M275: AN    DIX [AR2,P#0.0];
      JC    M277;
M276: LAR2  LD 24;
      L     DIB [AR2,P#0.0];
      INC   1;
      T     DIB [AR2,P#0.0];
      DEC   1;
      SLW   3;
      +AR2;
      L     DIB [AR1,P#0.0];
      T     DIB [AR2,P#0.0];
M277: L     LB 17;
M278: LOOP  M271;
      L     LB 28;
      JL    M279;
      JU    M135;
      JU    M131;
      JU    M130;
      JU    M054;
      JU    M053;
M279: NOP   0;
NETWORK
TITLE =
M280: CLR;
      LAR1  LD 0;
      L     DIW [AR1,P#18.0];
      SLD   3;
      T     LD 24;
      LAR2;
      LAR1;
      L     DIB [AR1,P#0.0];
      JU    M284;
M281: T     LB 17;
      +AR1  P#1.0;
      L     LB 14;
      L     DIB [AR1,P#0.0];
      <>I;
      JC    M282;
      L     DIB [LD 24];
      DEC   1;
      T     DIB [LD 24];
      JU    M283;
M282: +AR2  P#1.0;
      T     DIB [AR2,P#0.0];
M283: L     LB 17;
M284: LOOP  M281;
      A     L 29.0;
      JC    M162;
      JU    M150;
NETWORK
TITLE =
M285: L     DIB [AR1,P#0.0];
      JU    M287;
M286: T     LB 17;
      +AR1  P#1.0;
      L     DIB [AR1,P#0.0];
      SLW   7;
      LAR2  LD 0;
      +AR2;
      +AR2;
      L     B#16#0;
      T     DIB [AR2,P#0.0];
      L     LB 17;
M287: LOOP  M286;
      CLR;
      A     L 29.0;
      JC    M047;
      JU    M046;
NETWORK
TITLE =
M288: T     LW 20;
      LAR1  LD 4;
      L     DID [AR1,P#68.0];
      LAR1;
      CLR;
      A     L 29.0;
      JC    M289;
      LAR2  LD 0;
      L     DIB [AR2,P#26.0];
      SLW   3;
      +AR1;
M289: LAR2  LD 4;
      L     DID [AR2,P#80.0];
      LAR2;
      L     DIB [AR2,P#7.0];
      L     DIB [AR1,P#0.0];
      <I;
      LAR2  LD 4;
      S     DIX [AR2,P#26.5];
      JC    M290;
      INC   1;
      T     DIB [AR1,P#0.0];
      DEC   1;
      SLW   3;
      +AR1;
      L     LW 20;
      T     DIB [AR1,P#0.0];
M290: A     L 29.0;
      JC    M073;
      JU    M070;
NETWORK
TITLE =
// (network holds code this reader does not know; not shown)
NETWORK
TITLE =
M318: L     DINO;
      L     DID [AR1,P#52.0];
      +D;
      T     DID [AR1,P#52.0];
      SRD   16;
      T     LW 12;
      BLD   7;
      UC    "TIME_TCK";
      {     P#L 8.0 };
      BLD   8;
      L     LD 8;
      T     DID [AR1,P#18.0];
      L     LD 24;
      T     DID [AR1,P#80.0];
      LAR2;
      L     DID [AR1,P#48.0];
      AD    DW#16#7FFFF;
      T     LD 8;
      L     DID [AR1,P#36.0];
      +D;
      T     DID [AR1,P#36.0];
      TAK;
      L     DID [AR1,P#40.0];
      +D;
      T     DID [AR1,P#40.0];
      TAK;
      L     DID [AR1,P#44.0];
      +D;
      T     DID [AR1,P#44.0];
      TAK;
      L     DID [AR1,P#68.0];
      +D;
      T     DID [AR1,P#68.0];
      TAK;
      L     DID [AR1,P#28.0];
      +D;
      T     DID [AR1,P#28.0];
      T     LD 0;
      LAR1;
      A     L 29.1;
      JC    M321;
      L     W#16#FB;
      L     DIW [AR2,P#30.0];
      ==I;
      JC    M320;
      L     W#16#FC;
      ==I;
      JC    M319;
      L     DW#16#40000000;
      T     DID [AR2,P#14.0];
      L     DW#16#0;
      T     DID [AR2,P#18.0];
      L     B#16#2;
      JU    M322;
M319: L     DW#16#E000F6C8;
      T     DID [AR2,P#14.0];
      L     DW#16#E000800D;
      T     DID [AR2,P#18.0];
      L     B#16#A;
      JU    M322;
M320: L     DW#16#E3E0F6C8;
      T     DID [AR2,P#14.0];
      L     DW#16#E000BE0D;
      T     DID [AR2,P#18.0];
      L     B#16#A;
      JU    M322;
M321: L     DIW [AR2,P#32.0];
M322: L     LD 8;
      SRD   3;
      +D;
      T     DIW [AR1,P#12.0];
      TAR1;
      SRD   3;
      L     DIB [AR2,P#12.0];
      T     LB 14;
      INC   1;
      SLW   5;
      +D;
      L     DIW [AR2,P#0.0];
      SLD   2;
      +D;
      L     DIW [AR2,P#2.0];
      SLD   2;
      +D;
      T     DIW [AR1,P#14.0];
      L     DIB [AR2,P#9.0];
      T     LB 15;
      INC   2;
      SRW   1;
      SLW   1;
      T     DIB [AR1,P#2.0];
      L     LB 14;
      INC   2;
      SRW   1;
      SLW   1;
      T     DIB [AR1,P#3.0];
      L     DIB [AR2,P#6.0];
      INC   3;
      SRW   1;
      SLW   1;
      T     DIB [AR1,P#25.0];
      L     DIB [AR2,P#7.0];
      INC   3;
      SRW   1;
      SLW   1;
      T     DIB [AR1,P#26.0];
      L     LB 14;
      INC   3;
      SRW   1;
      SLW   1;
      T     DIB [AR1,P#27.0];
      L     LD 4;
      T     DID [AR1,P#8.0];
      L     DIW [AR1,P#14.0];
      L     DIB [AR1,P#25.0];
      SLW   1;
      +D;
      T     DIW [AR1,P#16.0];
      L     DIB [AR1,P#26.0];
      SLW   2;
      +D;
      SLD   3;
      T     DID [AR1,P#4.0];
      SRD   3;
      L     DIB [AR1,P#26.0];
      +D;
      T     DIW [AR1,P#18.0];
      TAR2;
      SRD   3;
      L     DIB [AR1,P#3.0];
      SLW   2;
      -D;
      T     DIW [AR1,P#22.0];
      L     DIB [AR1,P#2.0];
      SLW   2;
      -D;
      L     DIB [AR1,P#2.0];
      -D;
      T     DIW [AR1,P#20.0];
      L     DIB [AR1,P#26.0];
      -D;
      T     DIW [AR1,P#28.0];
      A     L 29.1;
      JC    M323;
      L     DIW [AR2,P#32.0];
      JU    M324;
M323: L     DIW [AR2,P#28.0];
M324: L     W#16#105;
      ==I;
      JC    M325;
      TAK;
      L     W#16#107;
      <>I;
      JC    M328;
M325: L     DIW [AR1,P#12.0];
      SLD   3;
      LAR2;
      L     B#16#0;
      L     LB 14;
M326: +AR1  P#32.0;
      TAK;
      INC   1;
      T     DIB [AR1,P#3.0];
      S     DIX [AR1,P#1.6];
      TAK;
      LOOP  M326;
      L     LB 15;
M327: +AR2  P#16.0;
      TAK;
      INC   1;
      T     DIB [AR2,P#3.0];
      S     DIX [AR2,P#0.3];
      TAK;
      LOOP  M327;
      LAR1  LD 0;
      L     B#16#7;
      T     DIB [AR1,P#30.0];
      LAR1  LD 4;
      L     DID [AR1,P#48.0];
      LAR2;
      UC    FB [LW 12];
M328: LAR1  LD 4;
      SET;
      S     DIX [AR1,P#27.2];
      JU    M005;
NETWORK
TITLE =
// (network holds code this reader does not know; not shown)
END_FUNCTION

FUNCTION "TE-ANEI" : VOID	// FC 78
AUTHOR : SIMATIC
FAMILY : EA_DIS
NAME : TE_ANEI
VERSION : 3.0
BEGIN
// (block stored without names or comments; labels and parameter names are numbered)
NETWORK
TITLE =
      L     #PARAM12;
      L     31;
      AW;
      T     MB 200;
      L     #PARAM4;
      T     MW 210;
      A     M 200.0;
      JC    M003;
      L     #PARAM3;
      T     MW 202;
      L     #PARAM1;
      L     W#16#4550;
      ==I;
      JC    M001;
      L     MB 203;
      SLW   3;
      LAR1;
      L     DBW [AR1,P#0.0];
      T     MW 204;
      JU    M002;
M001: NOP   0;
      L     MB 203;
      SLW   3;
      LAR1;
      L     DBW [AR1,P#0.0];
      T     MW 204;
M002: NOP   0;
M003: NOP   0;
NETWORK
TITLE =
      L     MW 210;
      L     2;
      ==I;
      JC    M004;
      JU    M007;
M004: A     M 200.0;
      JC    M008;
      L     MW 204;
      T     MW 240;
      AN    M 240.7;
      JC    M005;
      L     MW 240;
      NEGI;
      DTR;
      L     -1.000000e+00;
      *R;
      JU    M006;
M005: L     MW 240;
      DTR;
M006: T     MD 230;
      L     MD 230;
      L     1.000000e+01;
      /R;
      T     MD 238;
      L     MD 238;
      L     #PARAM7;
      -R;
      T     MD 218;
      L     #PARAM8;
      L     #PARAM7;
      -R;
      T     MD 242;
      L     MD 218;
      L     MD 242;
      /R;
      L     1.000000e+04;
      *R;
      T     MD 214;
      JU    M009;
M007: JU    M011;
M008: JU    M010;
M009: O(;
      L     MD 230;
      L     8.501000e+03;
      >=R;
      );
      O(;
      L     MD 230;
      L     1.000000e+04;
      >=R;
      );
      =     M 240.0;
      O(;
      L     -2.001000e+03;
      L     MD 230;
      >=R;
      );
      O(;
      L     -2.430000e+03;
      L     MD 230;
      >=R;
      );
      =     M 240.1;
      O(;
      L     -2.431000e+03;
      L     MD 230;
      >=R;
      );
      O(;
      L     -3.276800e+04;
      L     MD 230;
      >=R;
      );
      =     M 240.2;
      O(;
      L     MD 230;
      L     1.000000e+04;
      >=R;
      );
      O(;
      L     MD 230;
      L     3.276700e+04;
      >=R;
      );
      =     M 240.3;
      O(;
      L     MD 230;
      L     -2.000000e+03;
      >=R;
      );
      O(;
      L     MD 230;
      L     8.500000e+03;
      >=R;
      );
      =     M 240.4;
      O(;
      A     M 240.0;
      A     M 240.3;
      A     M 240.4;
      );
      O(;
      A     M 240.1;
      A     M 240.2;
      );
      =     M 200.6;
      A     M 200.3;
      A     M 200.6;
      =     M 200.7;
      L     MD 238;
      JU    M012;
M010: R     M 200.7;
      L     #PARAM6;
      T     MD 206;
      L     #PARAM7;
      -R;
      T     MD 244;
      L     #PARAM8;
      L     #PARAM7;
      -R;
      T     MD 248;
      L     MD 244;
      L     MD 248;
      /R;
      L     1.000000e+04;
      *R;
      T     MD 214;
      L     MD 206;
      JU    M014;
M011: JU    M015;
M012: AN    M 200.7;
      ON    M 200.1;
      JC    M013;
      JU    M014;
      L     1.000000e+04;
      T     MD 214;
      L     #PARAM8;
M013: AN    M 200.7;
      ON    M 200.2;
      JC    M014;
      L     0.000000e+00;
      T     MD 214;
      L     #PARAM7;
M014: T     #PARAM10;
      L     MD 214;
      T     #PARAM11;
      L     MB 200;
      T     #PARAM12;
M015: NOP   0;
NETWORK
TITLE =
      L     MW 210;
      L     4;
      ==I;
      JC    M016;
      JU    M020;
M016: A     M 200.0;
      JC    M021;
      L     MW 204;
      T     MW 240;
      AN    M 240.7;
      JC    M018;
M017: L     MW 240;
      NEGI;
      DTR;
      L     -1.000000e+00;
      *R;
      JU    M019;
M018: L     MW 240;
      L     32760;
      >I;
      JC    M017;
      L     MW 240;
      DTR;
M019: T     MD 230;
      L     2.764800e+04;
      /R;
      L     1.000000e+04;
      *R;
      T     MD 214;
      L     #PARAM8;
      L     #PARAM7;
      -R;
      L     1.000000e+04;
      /R;
      T     MD 218;
      L     MD 214;
      L     MD 218;
      *R;
      T     MD 234;
      L     #PARAM7;
      +R;
      T     MD 238;
      JU    M022;
M020: JU    M024;
M021: JU    M023;
M022: O(;
      L     MD 230;
      L     2.764900e+04;
      >=R;
      );
      O(;
      L     MD 230;
      L     3.251100e+04;
      >=R;
      );
      =     M 240.0;
      O(;
      L     -2.764900e+04;
      L     MD 230;
      >=R;
      );
      O(;
      L     -3.251200e+04;
      L     MD 230;
      >=R;
      );
      =     M 240.1;
      O(;
      L     -3.251300e+04;
      L     MD 230;
      >=R;
      );
      O(;
      L     -3.276800e+04;
      L     MD 230;
      >=R;
      );
      =     M 240.2;
      O(;
      L     MD 230;
      L     3.251200e+04;
      >=R;
      );
      O(;
      L     MD 230;
      L     3.276700e+04;
      >=R;
      );
      =     M 240.3;
      O(;
      L     MD 230;
      L     -2.764800e+04;
      >=R;
      );
      O(;
      L     MD 230;
      L     2.764800e+04;
      >=R;
      );
      =     M 240.4;
      O(;
      A     M 240.0;
      A     M 240.3;
      A     M 240.4;
      );
      O(;
      A     M 240.1;
      A     M 240.2;
      );
      =     M 200.6;
      A     M 200.3;
      A     M 200.6;
      =     M 200.7;
      L     MD 238;
      JU    M025;
M023: R     M 200.7;
      L     #PARAM6;
      T     MD 206;
      L     #PARAM7;
      -R;
      T     MD 244;
      L     #PARAM8;
      L     #PARAM7;
      -R;
      T     MD 248;
      L     MD 244;
      L     MD 248;
      /R;
      L     1.000000e+04;
      *R;
      T     MD 214;
      L     MD 206;
      JU    M027;
M024: JU    M028;
M025: AN    M 200.7;
      ON    M 200.1;
      JC    M026;
      JU    M027;
      L     1.000000e+04;
      T     MD 214;
      L     #PARAM8;
M026: AN    M 200.7;
      ON    M 200.2;
      JC    M027;
      L     0.000000e+00;
      T     MD 214;
      L     #PARAM7;
M027: T     #PARAM10;
      L     MD 214;
      T     #PARAM11;
      L     MB 200;
      T     #PARAM12;
M028: NOP   0;
NETWORK
TITLE =
      L     MW 210;
      L     6;
      ==I;
      JC    M029;
      JU    M033;
M029: A     M 200.0;
      JC    M034;
      L     MW 204;
      T     MW 240;
      AN    M 240.7;
      JC    M031;
M030: L     MW 240;
      NEGI;
      DTR;
      L     -1.000000e+00;
      *R;
      JU    M032;
M031: L     MW 240;
      L     32760;
      >I;
      JC    M030;
      L     MW 240;
      DTR;
M032: T     MD 230;
      L     2.764800e+04;
      /R;
      L     1.000000e+04;
      *R;
      T     MD 214;
      L     #PARAM8;
      L     #PARAM7;
      -R;
      L     1.000000e+04;
      /R;
      T     MD 218;
      L     MD 214;
      L     MD 218;
      *R;
      T     MD 234;
      L     #PARAM7;
      +R;
      T     MD 238;
      JU    M035;
M033: JU    M037;
M034: JU    M036;
M035: O(;
      L     MD 230;
      L     2.764900e+04;
      >=R;
      );
      O(;
      L     MD 230;
      L     3.251100e+04;
      >=R;
      );
      =     M 240.0;
      O(;
      L     -1.000000e+00;
      L     MD 230;
      >=R;
      );
      O(;
      L     -4.864000e+03;
      L     MD 230;
      >=R;
      );
      =     M 240.1;
      O(;
      L     -4.865000e+03;
      L     MD 230;
      >=R;
      );
      O(;
      L     -3.276800e+04;
      L     MD 230;
      >=R;
      );
      =     M 240.2;
      O(;
      L     MD 230;
      L     3.251200e+04;
      >=R;
      );
      O(;
      L     MD 230;
      L     3.276700e+04;
      >=R;
      );
      =     M 240.3;
      O(;
      L     MD 230;
      L     0.000000e+00;
      >=R;
      );
      O(;
      L     MD 230;
      L     2.764800e+04;
      >=R;
      );
      =     M 240.4;
      O(;
      A     M 240.0;
      A     M 240.3;
      A     M 240.4;
      );
      O(;
      A     M 240.1;
      A     M 240.2;
      );
      =     M 200.6;
      A     M 200.3;
      A     M 200.6;
      =     M 200.7;
      L     MD 238;
      JU    M038;
M036: R     M 200.7;
      L     #PARAM6;
      T     MD 206;
      L     #PARAM7;
      -R;
      T     MD 244;
      L     #PARAM8;
      L     #PARAM7;
      -R;
      T     MD 248;
      L     MD 244;
      L     MD 248;
      /R;
      L     1.000000e+04;
      *R;
      T     MD 214;
      L     MD 206;
      JU    M040;
M037: JU    M041;
M038: AN    M 200.7;
      ON    M 200.1;
      JC    M039;
      JU    M040;
      L     1.000000e+04;
      T     MD 214;
      L     #PARAM8;
M039: AN    M 200.7;
      ON    M 200.2;
      JC    M040;
      L     0.000000e+00;
      T     MD 214;
      L     #PARAM7;
M040: T     #PARAM10;
      L     MD 214;
      T     #PARAM11;
      L     MB 200;
      T     #PARAM12;
M041: NOP   0;
NETWORK
TITLE =
      L     MW 210;
      L     7;
      ==I;
      JC    M042;
      JU    M046;
M042: A     M 200.0;
      JC    M047;
      L     MW 204;
      T     MW 240;
      AN    M 240.7;
      JC    M044;
M043: L     MW 240;
      NEGI;
      DTR;
      L     -1.000000e+00;
      *R;
      JU    M045;
M044: L     MW 240;
      L     32760;
      >I;
      JC    M043;
      L     MW 240;
      DTR;
M045: T     MD 230;
      L     1.820000e+04;
      /R;
      L     1.000000e+04;
      *R;
      T     MD 214;
      L     #PARAM8;
      L     #PARAM7;
      -R;
      L     1.000000e+04;
      /R;
      T     MD 218;
      L     MD 214;
      L     MD 218;
      *R;
      T     MD 234;
      L     #PARAM7;
      +R;
      T     MD 238;
      JU    M048;
M046: JU    M050;
M047: JU    M049;
M048: O(;
      L     MD 230;
      L     1.820100e+04;
      >=R;
      );
      O(;
      L     MD 230;
      L     2.070000e+04;
      >=R;
      );
      =     M 240.0;
      O(;
      L     -1.000000e+00;
      L     MD 230;
      >=R;
      );
      O(;
      L     -1.200000e+03;
      L     MD 230;
      >=R;
      );
      =     M 240.1;
      L     -3.276800e+04;
      L     MD 230;
      >=R;
      =     M 240.2;
      L     MD 230;
      L     2.070100e+04;
      >=R;
      =     M 240.3;
      O(;
      L     MD 230;
      L     0.000000e+00;
      >=R;
      );
      O(;
      L     MD 230;
      L     1.820000e+04;
      >=R;
      );
      =     M 240.4;
      O(;
      A     M 240.0;
      A     M 240.3;
      A     M 240.4;
      );
      O(;
      A     M 240.1;
      A     M 240.2;
      );
      =     M 200.6;
      A     M 200.3;
      A     M 200.6;
      =     M 200.7;
      L     MD 238;
      JU    M051;
M049: R     M 200.7;
      L     #PARAM6;
      T     MD 206;
      L     #PARAM7;
      -R;
      T     MD 244;
      L     #PARAM8;
      L     #PARAM7;
      -R;
      T     MD 248;
      L     MD 244;
      L     MD 248;
      /R;
      L     1.000000e+04;
      *R;
      T     MD 214;
      L     MD 206;
      JU    M053;
M050: JU    M054;
M051: AN    M 200.7;
      ON    M 200.1;
      JC    M052;
      JU    M053;
      L     1.000000e+04;
      T     MD 214;
      L     #PARAM8;
M052: AN    M 200.7;
      ON    M 200.2;
      JC    M053;
      L     0.000000e+00;
      T     MD 214;
      L     #PARAM7;
M053: T     #PARAM10;
      L     MD 214;
      T     #PARAM11;
      L     MB 200;
      T     #PARAM12;
M054: NOP   0;
NETWORK
TITLE =
      L     MW 210;
      L     8;
      ==I;
      JC    M055;
      JU    M059;
M055: A     M 200.0;
      JC    M060;
      L     MW 204;
      T     MW 240;
      AN    M 240.7;
      JC    M057;
M056: L     MW 240;
      NEGI;
      DTR;
      L     -1.000000e+00;
      *R;
      JU    M058;
M057: L     MW 240;
      L     32760;
      >I;
      JC    M056;
      L     MW 240;
      DTR;
M058: T     MD 230;
      L     2.315000e+04;
      /R;
      L     1.000000e+04;
      *R;
      T     MD 214;
      L     #PARAM8;
      L     #PARAM7;
      -R;
      L     1.000000e+04;
      /R;
      T     MD 218;
      L     MD 214;
      L     MD 218;
      *R;
      T     MD 234;
      L     #PARAM7;
      +R;
      T     MD 238;
      JU    M061;
M059: JU    M063;
M060: JU    M062;
M061: O(;
      L     MD 230;
      L     2.500000e+04;
      >=R;
      );
      O(;
      L     MD 230;
      L     2.315100e+04;
      >=R;
      );
      =     M 240.0;
      O(;
      L     -1.000000e+00;
      L     MD 230;
      >=R;
      );
      O(;
      L     -1.200000e+03;
      L     MD 230;
      >=R;
      );
      =     M 240.1;
      L     -3.276800e+04;
      L     MD 230;
      >=R;
      =     M 240.2;
      L     MD 230;
      L     2.500100e+04;
      >=R;
      =     M 240.3;
      O(;
      L     MD 230;
      L     0.000000e+00;
      >=R;
      );
      O(;
      L     MD 230;
      L     2.315000e+04;
      >=R;
      );
      =     M 240.4;
      O(;
      A     M 240.0;
      A     M 240.3;
      A     M 240.4;
      );
      O(;
      A     M 240.1;
      A     M 240.2;
      );
      =     M 200.6;
      A     M 200.3;
      A     M 200.6;
      =     M 200.7;
      L     MD 238;
      JU    M064;
M062: R     M 200.7;
      L     #PARAM6;
      T     MD 206;
      L     #PARAM7;
      -R;
      T     MD 244;
      L     #PARAM8;
      L     #PARAM7;
      -R;
      T     MD 248;
      L     MD 244;
      L     MD 248;
      /R;
      L     1.000000e+04;
      *R;
      T     MD 214;
      L     MD 206;
      JU    M066;
M063: JU    M067;
M064: AN    M 200.7;
      ON    M 200.1;
      JC    M065;
      JU    M066;
      L     1.000000e+04;
      T     MD 214;
      L     #PARAM8;
M065: AN    M 200.7;
      ON    M 200.2;
      JC    M066;
      L     0.000000e+00;
      T     MD 214;
      L     #PARAM7;
M066: T     #PARAM10;
      L     MD 214;
      T     #PARAM11;
      L     MB 200;
      T     #PARAM12;
M067: NOP   0;
NETWORK
TITLE =
      L     MW 210;
      L     9;
      ==I;
      JC    M068;
      JU    M073;
M068: A     M 200.0;
      JC    M074;
      L     MW 204;
      T     MW 240;
      AN    M 240.7;
      JC    M070;
M069: L     MW 240;
      NEGI;
      DTR;
      L     -1.000000e+00;
      *R;
      JU    M071;
M070: L     MW 240;
      L     32760;
      >I;
      JC    M069;
      L     MW 240;
      DTR;
      JU    M072;
M071: T     MD 230;
      L     #PARAM7;
      L     1.000000e+01;
      *R;
      T     MD 242;
      L     MD 230;
      L     MD 242;
      -R;
      L     1.270000e+04;
      /R;
      L     1.000000e+04;
      *R;
      T     MD 214;
      L     #PARAM8;
      L     #PARAM7;
      -R;
      L     1.000000e+04;
      /R;
      T     MD 218;
      L     MD 214;
      L     MD 218;
      *R;
      T     MD 234;
      L     #PARAM7;
      +R;
      T     MD 238;
      JU    M075;
M072: T     MD 230;
      L     #PARAM7;
      L     -1.000000e+01;
      *R;
      T     MD 242;
      L     MD 230;
      L     MD 242;
      +R;
      L     1.270000e+04;
      /R;
      L     1.000000e+04;
      *R;
      T     MD 214;
      L     #PARAM8;
      L     #PARAM7;
      -R;
      L     1.000000e+04;
      /R;
      T     MD 218;
      L     MD 214;
      L     MD 218;
      *R;
      T     MD 234;
      L     #PARAM7;
      +R;
      T     MD 238;
      JU    M075;
M073: JU    M077;
M074: JU    M076;
M075: O(;
      L     MD 230;
      L     1.200000e+04;
      >=R;
      );
      O(;
      L     MD 230;
      L     1.000100e+04;
      >=R;
      );
      =     M 240.0;
      O(;
      L     -1.000000e+00;
      L     MD 230;
      >=R;
      );
      O(;
      L     -1.200000e+03;
      L     MD 230;
      >=R;
      );
      =     M 240.1;
      L     -3.276800e+04;
      L     MD 230;
      >=R;
      =     M 240.2;
      L     MD 230;
      L     2.500100e+04;
      >=R;
      =     M 240.3;
      O(;
      L     MD 230;
      L     -2.700000e+03;
      >=R;
      );
      O(;
      L     MD 230;
      L     1.000000e+04;
      >=R;
      );
      =     M 240.4;
      O(;
      A     M 240.0;
      A     M 240.3;
      A     M 240.4;
      );
      O(;
      A     M 240.1;
      A     M 240.2;
      );
      =     M 200.6;
      A     M 200.3;
      A     M 200.6;
      =     M 200.7;
      L     MD 238;
      JU    M078;
M076: R     M 200.7;
      L     #PARAM6;
      T     MD 206;
      L     #PARAM7;
      -R;
      T     MD 244;
      L     #PARAM8;
      L     #PARAM7;
      -R;
      T     MD 248;
      L     MD 244;
      L     MD 248;
      /R;
      L     1.000000e+04;
      *R;
      T     MD 214;
      L     MD 206;
      JU    M080;
M077: JU    M081;
M078: AN    M 200.7;
      ON    M 200.1;
      JC    M079;
      JU    M080;
      L     1.000000e+04;
      T     MD 214;
      L     #PARAM8;
M079: AN    M 200.7;
      ON    M 200.2;
      JC    M040;
      L     0.000000e+00;
      T     MD 214;
      L     #PARAM7;
M080: T     #PARAM10;
      L     MD 214;
      T     #PARAM11;
      L     MB 200;
      T     #PARAM12;
M081: NOP   0;
NETWORK
TITLE =
      L     MW 210;
      L     10;
      ==I;
      JC    M082;
      JU    M085;
M082: A     M 200.0;
      JC    M086;
      L     MW 204;
      T     MW 240;
      AN    M 240.7;
      JC    M083;
      L     MW 240;
      NEGI;
      DTR;
      L     -1.000000e+00;
      *R;
      JU    M084;
M083: L     MW 240;
      DTR;
M084: T     MD 230;
      L     MD 230;
      L     1.000000e+01;
      /R;
      T     MD 238;
      L     MD 238;
      L     #PARAM7;
      -R;
      T     MD 218;
      L     #PARAM8;
      L     #PARAM7;
      -R;
      T     MD 242;
      L     MD 218;
      L     MD 242;
      /R;
      L     1.000000e+04;
      *R;
      T     MD 214;
      JU    M087;
M085: JU    M089;
M086: JU    M088;
M087: O(;
      L     MD 230;
      L     1.200100e+04;
      >=R;
      );
      O(;
      L     MD 230;
      L     1.450000e+04;
      >=R;
      );
      =     M 240.0;
      L     -2.100000e+03;
      L     MD 230;
      >=R;
      =     M 240.1;
      L     -2.100000e+03;
      L     MD 230;
      >=R;
      =     M 240.2;
      L     MD 230;
      L     1.450100e+04;
      >=R;
      =     M 240.3;
      O(;
      L     MD 230;
      L     -2.100000e+03;
      >=R;
      );
      O(;
      L     MD 230;
      L     1.200000e+03;
      >=R;
      );
      =     M 240.4;
      O(;
      A     M 240.0;
      A     M 240.3;
      A     M 240.4;
      );
      O(;
      A     M 240.1;
      A     M 240.2;
      );
      =     M 200.6;
      A     M 200.3;
      A     M 200.6;
      =     M 200.7;
      L     MD 238;
      JU    M090;
M088: R     M 200.7;
      L     #PARAM6;
      T     MD 206;
      L     #PARAM7;
      -R;
      T     MD 244;
      L     #PARAM8;
      L     #PARAM7;
      -R;
      T     MD 248;
      L     MD 244;
      L     MD 248;
      /R;
      L     1.000000e+04;
      *R;
      T     MD 214;
      L     MD 206;
      JU    M092;
M089: JU    M093;
M090: AN    M 200.7;
      ON    M 200.1;
      JC    M091;
      JU    M092;
      L     1.000000e+04;
      T     MD 214;
      L     #PARAM8;
M091: AN    M 200.7;
      ON    M 200.2;
      JC    M092;
      L     0.000000e+00;
      T     MD 214;
      L     #PARAM7;
M092: T     #PARAM10;
      L     MD 214;
      T     #PARAM11;
      L     MB 200;
      T     #PARAM12;
M093: NOP   0;
NETWORK
TITLE =
      L     MW 210;
      L     11;
      ==I;
      JC    M094;
      JU    M097;
M094: A     M 200.0;
      JC    M098;
      L     MW 204;
      T     MW 240;
      AN    M 240.7;
      JC    M095;
      L     MW 240;
      NEGI;
      DTR;
      L     -1.000000e+00;
      *R;
      JU    M096;
M095: L     MW 240;
      DTR;
M096: T     MD 230;
      L     MD 230;
      L     1.000000e+01;
      /R;
      T     MD 238;
      L     MD 238;
      L     #PARAM7;
      -R;
      T     MD 218;
      L     #PARAM8;
      L     #PARAM7;
      -R;
      T     MD 242;
      L     MD 218;
      L     MD 242;
      /R;
      L     1.000000e+04;
      *R;
      T     MD 214;
      JU    M099;
M097: JU    M101;
M098: JU    M100;
M099: O(;
      L     MD 230;
      L     1.666200e+04;
      >=R;
      );
      O(;
      L     MD 230;
      L     1.372100e+04;
      >=R;
      );
      =     M 240.0;
      L     -2.700000e+03;
      L     MD 230;
      >=R;
      =     M 240.1;
      L     -2.700000e+03;
      L     MD 230;
      >=R;
      =     M 240.2;
      L     MD 230;
      L     1.622100e+04;
      >=R;
      =     M 240.3;
      O(;
      L     MD 230;
      L     -2.700000e+03;
      >=R;
      );
      O(;
      L     MD 230;
      L     1.372000e+03;
      >=R;
      );
      =     M 240.4;
      O(;
      A     M 240.0;
      A     M 240.3;
      A     M 240.4;
      );
      O(;
      A     M 240.1;
      A     M 240.2;
      );
      =     M 200.6;
      A     M 200.3;
      A     M 200.6;
      =     M 200.7;
      L     MD 238;
      JU    M102;
M100: R     M 200.7;
      L     #PARAM6;
      T     MD 206;
      L     #PARAM7;
      -R;
      T     MD 244;
      L     #PARAM8;
      L     #PARAM7;
      -R;
      T     MD 248;
      L     MD 244;
      L     MD 248;
      /R;
      L     1.000000e+04;
      *R;
      T     MD 214;
      L     MD 206;
      JU    M104;
M101: JU    M105;
M102: AN    M 200.7;
      ON    M 200.1;
      JC    M103;
      JU    M104;
      L     1.000000e+04;
      T     MD 214;
      L     #PARAM8;
M103: AN    M 200.7;
      ON    M 200.2;
      JC    M104;
      L     0.000000e+00;
      T     MD 214;
      L     #PARAM7;
M104: T     #PARAM10;
      L     MD 214;
      T     #PARAM11;
      L     MB 200;
      T     #PARAM12;
M105: NOP   0;
NETWORK
TITLE =
      L     MW 210;
      L     12;
      ==I;
      JC    M106;
      JU    M109;
M106: A     M 200.0;
      JC    M110;
      L     MW 204;
      T     MW 240;
      AN    M 240.7;
      JC    M107;
      L     MW 240;
      NEGI;
      DTR;
      L     -1.000000e+00;
      *R;
      JU    M108;
M107: L     MW 240;
      DTR;
M108: T     MD 230;
      L     MD 230;
      L     1.000000e+01;
      /R;
      T     MD 238;
      L     MD 238;
      L     #PARAM7;
      -R;
      T     MD 218;
      L     #PARAM8;
      L     #PARAM7;
      -R;
      T     MD 242;
      L     MD 218;
      L     MD 242;
      /R;
      L     1.000000e+04;
      *R;
      T     MD 214;
      JU    M111;
M109: JU    M113;
M110: JU    M112;
M111: O(;
      L     MD 230;
      L     1.150000e+04;
      >=R;
      );
      O(;
      L     MD 230;
      L     9.001000e+03;
      >=R;
      );
      =     M 240.0;
      L     -2.000000e+03;
      L     MD 230;
      >=R;
      =     M 240.1;
      L     -2.000000e+03;
      L     MD 230;
      >=R;
      =     M 240.2;
      L     MD 230;
      L     9.001000e+03;
      >=R;
      =     M 240.3;
      O(;
      L     MD 230;
      L     -2.000000e+03;
      >=R;
      );
      O(;
      L     MD 230;
      L     9.000000e+03;
      >=R;
      );
      =     M 240.4;
      O(;
      A     M 240.0;
      A     M 240.3;
      A     M 240.4;
      );
      O(;
      A     M 240.1;
      A     M 240.2;
      );
      =     M 200.6;
      A     M 200.3;
      A     M 200.6;
      =     M 200.7;
      L     MD 238;
      JU    M114;
M112: R     M 200.7;
      L     #PARAM6;
      T     MD 206;
      L     #PARAM7;
      -R;
      T     MD 244;
      L     #PARAM8;
      L     #PARAM7;
      -R;
      T     MD 248;
      L     MD 244;
      L     MD 248;
      /R;
      L     1.000000e+04;
      *R;
      T     MD 214;
      L     MD 206;
      JU    M116;
M113: JU    M117;
M114: AN    M 200.7;
      ON    M 200.1;
      JC    M115;
      JU    M116;
      L     1.000000e+04;
      T     MD 214;
      L     #PARAM8;
M115: AN    M 200.7;
      ON    M 200.2;
      JC    M116;
      L     0.000000e+00;
      T     MD 214;
      L     #PARAM7;
M116: T     #PARAM10;
      L     MD 214;
      T     #PARAM11;
      L     MB 200;
      T     #PARAM12;
M117: NOP   0;
NETWORK
TITLE =
      L     MW 210;
      L     12;
      ==I;
      JC    M118;
      JU    M121;
M118: A     M 200.0;
      JC    M122;
      L     MW 204;
      T     MW 240;
      AN    M 240.7;
      JC    M119;
      L     MW 240;
      NEGI;
      DTR;
      L     -1.000000e+00;
      *R;
      JU    M120;
M119: L     MW 240;
      DTR;
M120: T     MD 230;
      L     MD 230;
      L     1.000000e+01;
      /R;
      T     MD 238;
      L     MD 238;
      L     #PARAM7;
      -R;
      T     MD 218;
      L     #PARAM8;
      L     #PARAM7;
      -R;
      T     MD 242;
      L     MD 218;
      L     MD 242;
      /R;
      L     1.000000e+04;
      *R;
      T     MD 214;
      JU    M123;
M121: JU    M125;
M122: JU    M124;
M123: O(;
      L     MD 230;
      L     1.550000e+04;
      >=R;
      );
      O(;
      L     MD 230;
      L     1.300100e+04;
      >=R;
      );
      =     M 240.0;
      L     -2.700000e+03;
      L     MD 230;
      >=R;
      =     M 240.1;
      L     -2.700000e+03;
      L     MD 230;
      >=R;
      =     M 240.2;
      L     MD 230;
      L     1.550100e+04;
      >=R;
      =     M 240.3;
      O(;
      L     MD 230;
      L     -2.700000e+03;
      >=R;
      );
      O(;
      L     MD 230;
      L     1.550000e+03;
      >=R;
      );
      =     M 240.4;
      O(;
      A     M 240.0;
      A     M 240.3;
      A     M 240.4;
      );
      O(;
      A     M 240.1;
      A     M 240.2;
      );
      =     M 200.6;
      A     M 200.3;
      A     M 200.6;
      =     M 200.7;
      L     MD 238;
      JU    M126;
M124: R     M 200.7;
      L     #PARAM6;
      T     MD 206;
      L     #PARAM7;
      -R;
      T     MD 244;
      L     #PARAM8;
      L     #PARAM7;
      -R;
      T     MD 248;
      L     MD 244;
      L     MD 248;
      /R;
      L     1.000000e+04;
      *R;
      T     MD 214;
      L     MD 206;
      JU    M128;
M125: JU    M129;
M126: AN    M 200.7;
      ON    M 200.1;
      JC    M127;
      JU    M128;
      L     1.000000e+04;
      T     MD 214;
      L     #PARAM8;
M127: AN    M 200.7;
      ON    M 200.2;
      JC    M128;
      L     0.000000e+00;
      T     MD 214;
      L     #PARAM7;
M128: T     #PARAM10;
      L     MD 214;
      T     #PARAM11;
      L     MB 200;
      T     #PARAM12;
M129: NOP   0;
NETWORK
TITLE =
      L     MW 210;
      L     14;
      ==I;
      JC    M130;
      JU    M133;
M130: A     M 200.0;
      JC    M134;
      L     MW 204;
      T     MW 240;
      AN    M 240.7;
      JC    M131;
      L     MW 240;
      NEGI;
      DTR;
      L     -1.000000e+00;
      *R;
      JU    M132;
M131: L     MW 240;
      DTR;
M132: T     MD 230;
      L     MD 230;
      L     1.000000e+01;
      /R;
      T     MD 238;
      L     MD 238;
      L     #PARAM7;
      -R;
      T     MD 218;
      L     #PARAM8;
      L     #PARAM7;
      -R;
      T     MD 242;
      L     MD 218;
      L     MD 242;
      /R;
      L     1.000000e+04;
      *R;
      T     MD 214;
      JU    M135;
M133: JU    M137;
M134: JU    M136;
M135: O(;
      L     MD 230;
      L     2.019000e+04;
      >=R;
      );
      O(;
      L     MD 230;
      L     1.769100e+04;
      >=R;
      );
      =     M 240.0;
      O(;
      L     -5.010000e+02;
      L     MD 230;
      >=R;
      );
      O(;
      L     -1.700000e+03;
      L     MD 230;
      >=R;
      );
      =     M 240.1;
      O(;
      L     2.090100e+04;
      L     MD 230;
      >=R;
      );
      O(;
      L     -1.200000e+03;
      L     MD 230;
      >=R;
      );
      =     M 240.2;
      O(;
      L     -1.000000e+00;
      L     MD 230;
      >=R;
      );
      O(;
      L     -1.200000e+03;
      L     MD 230;
      >=R;
      );
      =     M 240.3;
      O(;
      L     MD 230;
      L     -5.000000e+02;
      >=R;
      );
      O(;
      L     MD 230;
      L     1.769000e+04;
      >=R;
      );
      =     M 240.4;
      O(;
      A     M 240.0;
      A     M 240.3;
      A     M 240.4;
      );
      O(;
      A     M 240.1;
      A     M 240.2;
      );
      =     M 200.6;
      A     M 200.3;
      A     M 200.6;
      =     M 200.7;
      L     MD 238;
      JU    M138;
M136: R     M 200.7;
      L     #PARAM6;
      T     MD 206;
      L     #PARAM7;
      -R;
      T     MD 244;
      L     #PARAM8;
      L     #PARAM7;
      -R;
      T     MD 248;
      L     MD 244;
      L     MD 248;
      /R;
      L     1.000000e+04;
      *R;
      T     MD 214;
      L     MD 206;
      JU    M140;
M137: JU    M141;
M138: AN    M 200.7;
      ON    M 200.1;
      JC    M139;
      JU    M140;
      L     1.000000e+04;
      T     MD 214;
      L     #PARAM8;
M139: AN    M 200.7;
      ON    M 200.2;
      JC    M140;
      L     0.000000e+00;
      T     MD 214;
      L     #PARAM7;
M140: T     #PARAM10;
      L     MD 214;
      T     #PARAM11;
      L     MB 200;
      T     #PARAM12;
M141: NOP   0;
NETWORK
TITLE =
      L     MW 210;
      L     14;
      ==I;
      JC    M142;
      JU    M145;
M142: A     M 200.0;
      JC    M146;
      L     MW 204;
      T     MW 240;
      AN    M 240.7;
      JC    M143;
      L     MW 240;
      NEGI;
      DTR;
      L     -1.000000e+00;
      *R;
      JU    M144;
M143: L     MW 240;
      DTR;
M144: T     MD 230;
      L     MD 230;
      L     1.000000e+01;
      /R;
      T     MD 238;
      L     MD 238;
      L     #PARAM7;
      -R;
      T     MD 218;
      L     #PARAM8;
      L     #PARAM7;
      -R;
      T     MD 242;
      L     MD 218;
      L     MD 242;
      /R;
      L     1.000000e+04;
      *R;
      T     MD 214;
      JU    M147;
M145: JU    M149;
M146: JU    M148;
M147: O(;
      L     MD 230;
      L     1.666200e+04;
      >=R;
      );
      O(;
      L     MD 230;
      L     1.372100e+04;
      >=R;
      );
      =     M 240.0;
      L     -2.700000e+03;
      L     MD 230;
      >=R;
      =     M 240.1;
      L     -2.700000e+03;
      L     MD 230;
      >=R;
      =     M 240.2;
      L     MD 230;
      L     1.622100e+04;
      >=R;
      =     M 240.3;
      O(;
      L     MD 230;
      L     -2.700000e+03;
      >=R;
      );
      O(;
      L     MD 230;
      L     1.372000e+03;
      >=R;
      );
      =     M 240.4;
      O(;
      A     M 240.0;
      A     M 240.3;
      A     M 240.4;
      );
      O(;
      A     M 240.1;
      A     M 240.2;
      );
      =     M 200.6;
      A     M 200.3;
      A     M 200.6;
      =     M 200.7;
      L     MD 238;
      JU    M150;
M148: R     M 200.7;
      L     #PARAM6;
      T     MD 206;
      L     #PARAM7;
      -R;
      T     MD 244;
      L     #PARAM8;
      L     #PARAM7;
      -R;
      T     MD 248;
      L     MD 244;
      L     MD 248;
      /R;
      L     1.000000e+04;
      *R;
      T     MD 214;
      L     MD 206;
      JU    M152;
M149: JU    M153;
M150: AN    M 200.7;
      ON    M 200.1;
      JC    M151;
      JU    M152;
      L     1.000000e+04;
      T     MD 214;
      L     #PARAM8;
M151: AN    M 200.7;
      ON    M 200.2;
      JC    M152;
      L     0.000000e+00;
      T     MD 214;
      L     #PARAM7;
M152: T     #PARAM10;
      L     MD 214;
      T     #PARAM11;
      L     MB 200;
      T     #PARAM12;
M153: NOP   0;
NETWORK
TITLE =
      L     0;
      L     #PARAM9;
      ==I;
      BEC;
      T     MW 206;
      T     MW 220;
      L     MB 206;
      SLW   3;
      LAR1;
      L     DBW [AR1,P#0.0];
      T     MW 208;
      L     MW 220;
      SLW   12;
      SRW   12;
      T     MW 220;
      L     8;
      L     MB 221;
      >I;
      JC    M154;
      +     -8;
      SLW   8;
      INC   208;
      JU    M155;
M154: SLW   8;
      INC   209;
M155: T     MW 210;
      L     MB 210;
      L     MB 211;
      SLW   3;
      OW;
      LAR2;
      A     M 200.7;
      =     M [AR2,P#0.0];
      L     MB 206;
      SLW   3;
      LAR1;
      L     MW 208;
      T     DBW [AR1,P#0.0];
END_FUNCTION

FUNCTION "TE-ANAU" : VOID	// FC 79
AUTHOR : SIMATIC
FAMILY : EA_DIS
NAME : TE_ANAU
VERSION : 3.0
BEGIN
// (block stored without names or comments; labels and parameter names are numbered)
NETWORK
TITLE =
      L     #PARAM1;
      T     MB 255;
      L     #PARAM3;
      T     MB 254;
      L     1;
      >I;
      JC    M001;
      L     #PARAM2;
      L     2.764800e+00;
      *R;
      RND;
      T     MW 240;
      JU    M004;
M001: L     #PARAM2;
      L     0.000000e+00;
      <R;
      JC    M002;
      TAK;
      L     2.764800e+00;
      *R;
      T     MD 250;
      JU    M003;
M002: TAK;
      L     -1.000000e+00;
      *R;
M003: RND;
      T     MW 240;
M004: A     M 255.1;
      JC    M005;
      L     MW 240;
      T     #PARAM4;
M005: NOP   0;
END_FUNCTION

// FC 105: know-how protected block, not included

FUNCTION "FC 110" : VOID	// FC 110
VERSION : 0.1
BEGIN
// (block stored without names or comments; labels and parameter names are numbered)
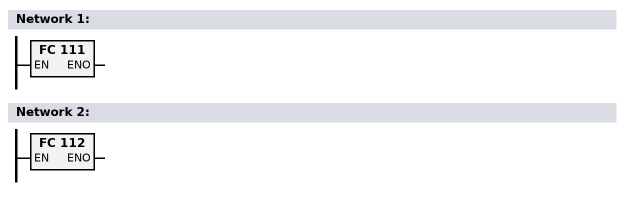
NETWORK
TITLE =
      CALL  "FC 111";
      NOP   0;
NETWORK
TITLE =
      CALL  "FC 112";
      NOP   0;
END_FUNCTION

FUNCTION "FC 111" : VOID	// FC 111
VERSION : 0.1
BEGIN
// (block stored without names or comments; labels and parameter names are numbered)
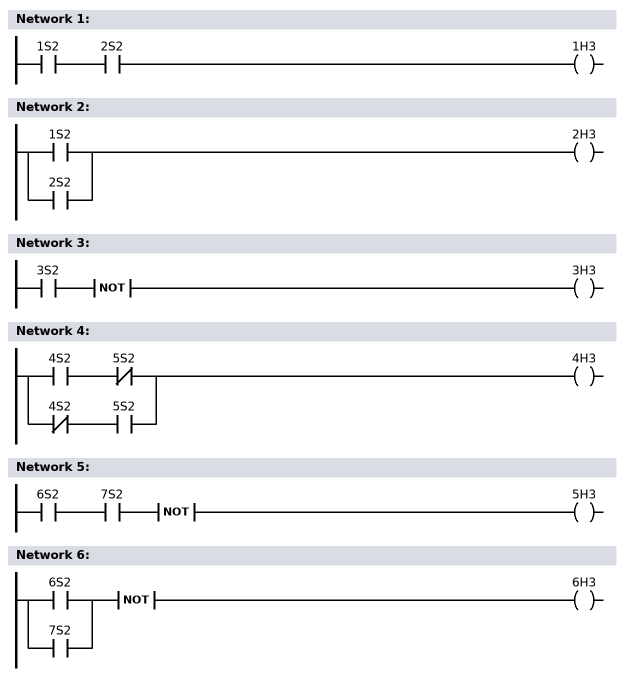
NETWORK
TITLE =
      A     "1S2";
      A     "2S2";
      =     "1H3";
NETWORK
TITLE =
      O     "1S2";
      O     "2S2";
      =     "2H3";
NETWORK
TITLE =
      A     "3S2";
      NOT;
      =     "3H3";
NETWORK
TITLE =
      A     "4S2";
      AN    "5S2";
      O;
      AN    "4S2";
      A     "5S2";
      =     "4H3";
NETWORK
TITLE =
      A     "6S2";
      A     "7S2";
      NOT;
      =     "5H3";
NETWORK
TITLE =
      A(;
      O     "6S2";
      O     "7S2";
      );
      NOT;
      =     "6H3";
END_FUNCTION

FUNCTION "FC 112" : VOID	// FC 112
VERSION : 0.1
BEGIN
// (block stored without names or comments; labels and parameter names are numbered)
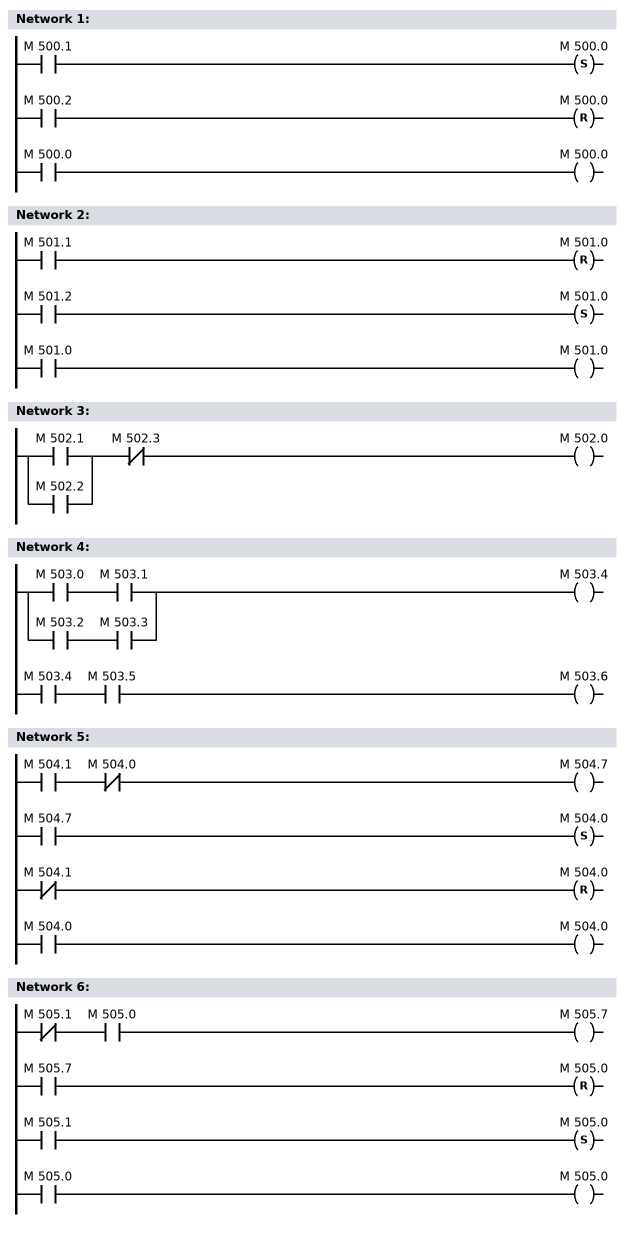
NETWORK
TITLE =
      A     M 500.1;
      S     M 500.0;
      A     M 500.2;
      R     M 500.0;
      A     M 500.0;
      =     M 500.0;
NETWORK
TITLE =
      A     M 501.1;
      R     M 501.0;
      A     M 501.2;
      S     M 501.0;
      A     M 501.0;
      =     M 501.0;
NETWORK
TITLE =
      A(;
      O     M 502.1;
      O     M 502.2;
      );
      AN    M 502.3;
      =     M 502.0;
NETWORK
TITLE =
      A(;
      A     M 503.0;
      A     M 503.1;
      O;
      A     M 503.2;
      A     M 503.3;
      );
      =     M 503.4;
      A     M 503.4;
      A     M 503.5;
      =     M 503.6;
NETWORK
TITLE =
      A     M 504.1;
      AN    M 504.0;
      =     M 504.7;
      A     M 504.7;
      S     M 504.0;
      AN    M 504.1;
      R     M 504.0;
      A     M 504.0;
      =     M 504.0;
NETWORK
TITLE =
      AN    M 505.1;
      A     M 505.0;
      =     M 505.7;
      A     M 505.7;
      R     M 505.0;
      A     M 505.1;
      S     M 505.0;
      A     M 505.0;
      =     M 505.0;
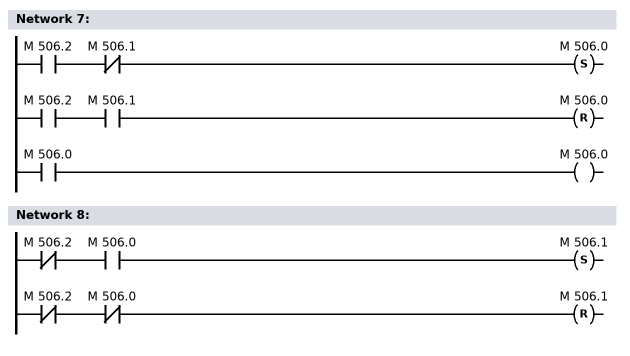
NETWORK
TITLE =
      A     M 506.2;
      AN    M 506.1;
      S     M 506.0;
      A     M 506.2;
      A     M 506.1;
      R     M 506.0;
      A     M 506.0;
      =     M 506.0;
NETWORK
TITLE =
      AN    M 506.2;
      A     M 506.0;
      S     M 506.1;
      AN    M 506.2;
      AN    M 506.0;
      R     M 506.1;
      NOP   0;
END_FUNCTION

FUNCTION "FC 113" : VOID	// FC 113
VERSION : 0.1
BEGIN
// (block stored without names or comments; labels and parameter names are numbered)
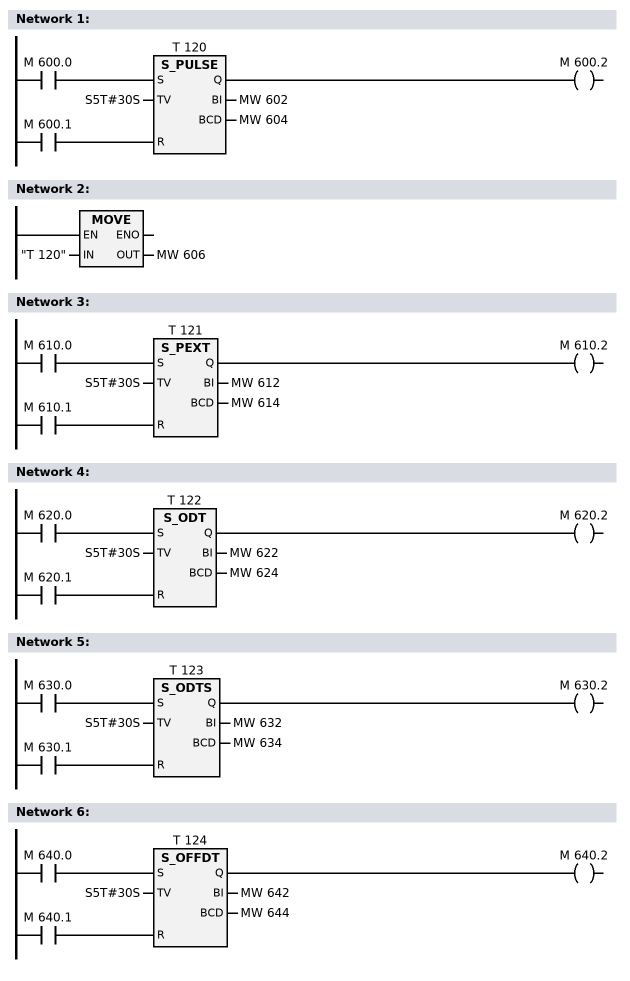
NETWORK
TITLE =
      A     M 600.0;
      L     S5T#30S;
      SP    "T 120";
      A     M 600.1;
      R     "T 120";
      L     "T 120";
      T     MW 602;
      LC    "T 120";
      T     MW 604;
      A     "T 120";
      =     M 600.2;
NETWORK
TITLE =
      L     "T 120";
      T     MW 606;
      NOP   0;
NETWORK
TITLE =
      A     M 610.0;
      L     S5T#30S;
      SE    "T 121";
      A     M 610.1;
      R     "T 121";
      L     "T 121";
      T     MW 612;
      LC    "T 121";
      T     MW 614;
      A     "T 121";
      =     M 610.2;
NETWORK
TITLE =
      A     M 620.0;
      L     S5T#30S;
      SD    "T 122";
      A     M 620.1;
      R     "T 122";
      L     "T 122";
      T     MW 622;
      LC    "T 122";
      T     MW 624;
      A     "T 122";
      =     M 620.2;
NETWORK
TITLE =
      A     M 630.0;
      L     S5T#30S;
      SS    "T 123";
      A     M 630.1;
      R     "T 123";
      L     "T 123";
      T     MW 632;
      LC    "T 123";
      T     MW 634;
      A     "T 123";
      =     M 630.2;
NETWORK
TITLE =
      A     M 640.0;
      L     S5T#30S;
      SF    "T 124";
      A     M 640.1;
      R     "T 124";
      L     "T 124";
      T     MW 642;
      LC    "T 124";
      T     MW 644;
      A     "T 124";
      =     M 640.2;
END_FUNCTION

FUNCTION "FC 114" : VOID	// FC 114
VERSION : 0.1
BEGIN
// (block stored without names or comments; labels and parameter names are numbered)
NETWORK
TITLE =
      A     M 700.0;
      CU    "Z 120";
      A     M 700.1;
      CD    "Z 120";
      A     M 700.2;
      L     MW 702;
      S     "Z 120";
      A     M 700.3;
      R     "Z 120";
      L     "Z 120";
      T     MW 704;
      LC    "Z 120";
      T     MW 706;
      A     "Z 120";
      =     M 700.4;
NETWORK
TITLE =
      A     M 710.0;
      CU    "Z 121";
      BLD   101;
      A     M 710.2;
      L     MW 712;
      S     "Z 121";
      A     M 710.3;
      R     "Z 121";
      L     "Z 121";
      T     MW 714;
      LC    "Z 121";
      T     MW 716;
      A     "Z 121";
      =     M 710.4;
NETWORK
TITLE =
      A     M 720.0;
      CD    "Z 122";
      BLD   101;
      A     M 720.2;
      L     MW 722;
      S     "Z 122";
      A     M 720.3;
      R     "Z 122";
      L     "Z 122";
      T     MW 724;
      LC    "Z 122";
      T     MW 726;
      A     "Z 122";
      =     M 720.4;
END_FUNCTION

FUNCTION FC 118 : VOID
VERSION : 0.1
BEGIN
// (block stored without names or comments; labels and parameter names are numbered)
NETWORK
TITLE =
      AN    "M 118.1";
      =     "M 118.0";
NETWORK
TITLE =
      CALL  SFC 67 (
           $1                       := P#M 118.0,
           $2                       := TRUE,
           $3                       := 3,
           $4                       := P#DB118.DBX 14.0 BYTE 12,
           $5                       := DB118.DBW 12,
           $6                       := "M 118.1",
           $7                       := P#DB118.DBX 0.0 BYTE 12);
NETWORK
TITLE =
NETWORK
TITLE =
      AN    M 118.3;
      =     M 118.2;
NETWORK
TITLE =
      CALL  SFC 68 (
           $1                       := M 118.2,
           $2                       := TRUE,
           $3                       := 3,
           $4                       := P#DB118.DBX 14.0 BYTE 12,
           $5                       := P#DB118.DBX 0.0 BYTE 12,
           $6                       := DB118.DBW 26,
           $7                       := M 118.3);
NETWORK
TITLE =
NETWORK
TITLE =
      A     DB118.DBX 1.7;
      =     DB118.DBX 15.7;
NETWORK
TITLE =
      A     DB118.DBX 1.7;
      FP    M 118.5;
      =     M 118.6;
NETWORK
TITLE =
      A     M 118.6;
      L     S5T#3S;
      SE    "T 118";
NETWORK
TITLE =
      A     "T 118";
      =     M 118.7;
NETWORK
TITLE =
      AN    M 118.7;
      JNB   M001;
      SET;
      R     DB118.DBX 0.0;
      R     DB118.DBX 0.1;
      R     DB118.DBX 0.2;
      R     DB118.DBX 0.3;
      R     DB118.DBX 0.4;
      R     DB118.DBX 0.5;
      R     DB118.DBX 0.6;
      R     DB118.DBX 0.7;
      R     DB118.DBX 1.0;
      R     DB118.DBX 1.1;
      R     DB118.DBX 1.2;
      R     DB118.DBX 1.3;
      R     DB118.DBX 1.4;
      R     DB118.DBX 1.5;
      R     DB118.DBX 1.6;
      L     0;
      T     DB118.DBD 4;
      T     DB118.DBD 8;
M001: NOP   0;
NETWORK
TITLE =
      BE;
END_FUNCTION

FUNCTION "FC 120" : VOID	// FC 120
VERSION : 0.1
BEGIN
// (block stored without names or comments; labels and parameter names are numbered)
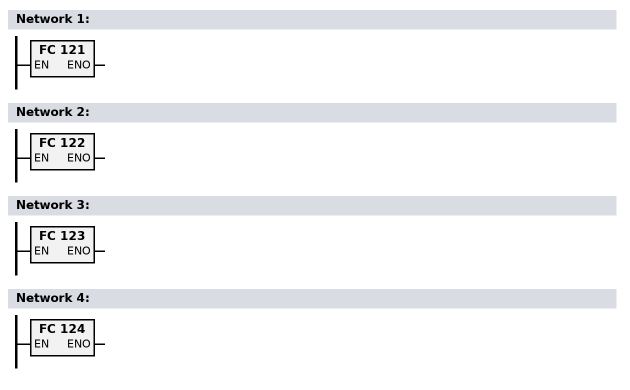
NETWORK
TITLE =
      CALL  "FC 121";
      NOP   0;
NETWORK
TITLE =
      CALL  "FC 122";
      NOP   0;
NETWORK
TITLE =
      CALL  "FC 123";
      NOP   0;
NETWORK
TITLE =
      CALL  "FC 124";
      NOP   0;
END_FUNCTION

FUNCTION "FC 121" : VOID	// FC 121
VERSION : 0.1
BEGIN
// (block stored without names or comments; labels and parameter names are numbered)
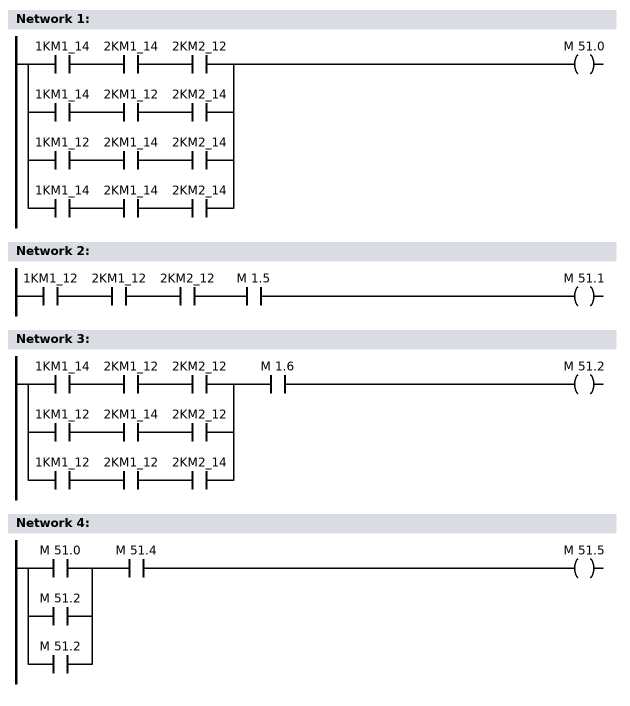
NETWORK
TITLE =
      A     "1KM1_14";
      A     "2KM1_14";
      A     "2KM2_12";
      O;
      A     "1KM1_14";
      A     "2KM1_12";
      A     "2KM2_14";
      O;
      A     "1KM1_12";
      A     "2KM1_14";
      A     "2KM2_14";
      O;
      A     "1KM1_14";
      A     "2KM1_14";
      A     "2KM2_14";
      =     "M 51.0";
NETWORK
TITLE =
      A     "1KM1_12";
      A     "2KM1_12";
      A     "2KM2_12";
      A     "M 1.5";
      =     "M 51.1";
NETWORK
TITLE =
      A(;
      A     "1KM1_14";
      A     "2KM1_12";
      A     "2KM2_12";
      O;
      A     "1KM1_12";
      A     "2KM1_14";
      A     "2KM2_12";
      O;
      A     "1KM1_12";
      A     "2KM1_12";
      A     "2KM2_14";
      );
      A     "M 1.6";
      =     "M 51.2";
NETWORK
TITLE =
      A(;
      O     "M 51.0";
      O     "M 51.2";
      O     "M 51.2";
      );
      A     "M 51.4";
      =     "M 51.5";
END_FUNCTION

FUNCTION "FC 122" : VOID	// FC 122
VERSION : 0.1
BEGIN
// (block stored without names or comments; labels and parameter names are numbered)
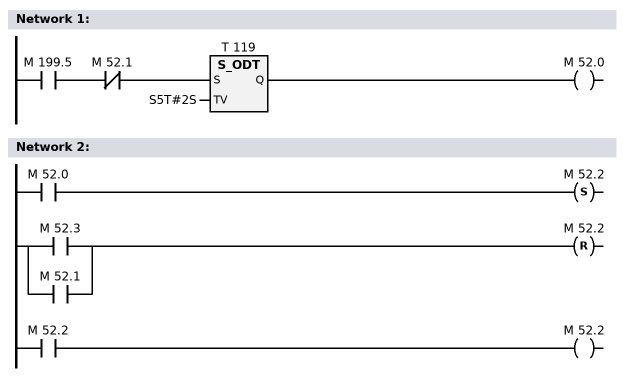
NETWORK
TITLE =
      A     "M 199.5";
      AN    "M 52.1";
      L     S5T#2S;
      SD    "T 119";
      NOP   0;
      NOP   0;
      NOP   0;
      A     "T 119";
      =     "M 52.0";
NETWORK
TITLE =
      A     "M 52.0";
      S     "M 52.2";
      A(;
      O     "M 52.3";
      O     "M 52.1";
      );
      R     "M 52.2";
      A     "M 52.2";
      =     "M 52.2";
END_FUNCTION

FUNCTION "FC 123" : VOID	// FC 123
VERSION : 0.1
BEGIN
// (block stored without names or comments; labels and parameter names are numbered)
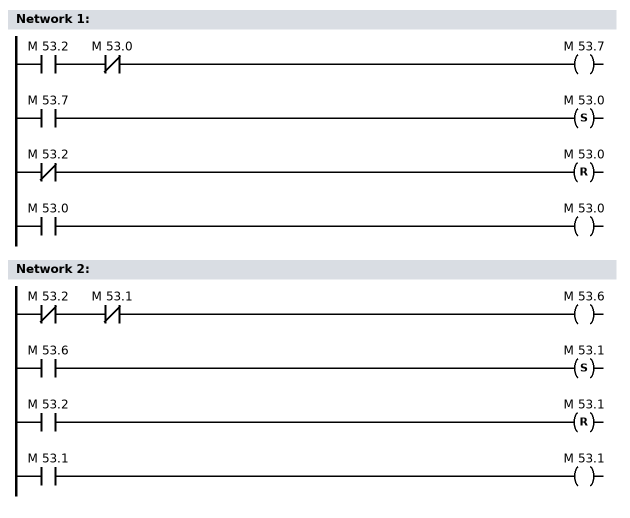
NETWORK
TITLE =
      A     "M 53.2";
      AN    "M 53.0";
      =     "M 53.7";
      A     "M 53.7";
      S     "M 53.0";
      AN    "M 53.2";
      R     "M 53.0";
      A     "M 53.0";
      =     "M 53.0";
NETWORK
TITLE =
      AN    "M 53.2";
      AN    "M 53.1";
      =     "M 53.6";
      A     "M 53.6";
      S     "M 53.1";
      A     "M 53.2";
      R     "M 53.1";
      A     "M 53.1";
      =     "M 53.1";
NETWORK
TITLE =
      A     "M 53.3";
      A     "M 53.7";
      CU    "Z 119";
      A     "M 53.3";
      A     "M 53.6";
      CD    "Z 119";
      A     "M 53.5";
      L     "MW 54";
      S     "Z 119";
      NOP   0;
      NOP   0;
      LC    "Z 119";
      T     "MW 56";
      A     "Z 119";
      =     "M 53.4";
END_FUNCTION

FUNCTION "FC 124" : VOID	// FC 124
VERSION : 0.1
BEGIN
// (block stored without names or comments; labels and parameter names are numbered)
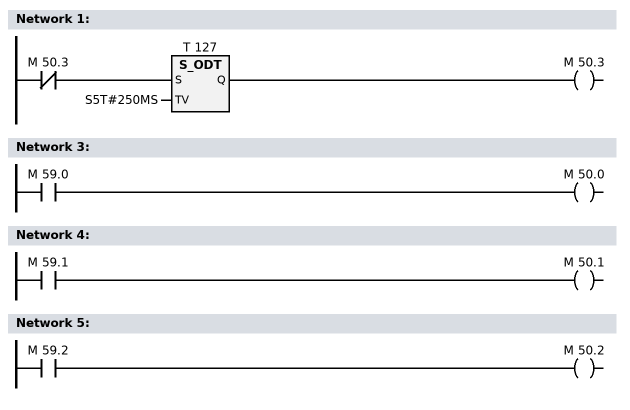
NETWORK
TITLE =
      AN    "M 50.3";
      L     S5T#250MS;
      SD    "T 127";
      NOP   0;
      NOP   0;
      NOP   0;
      A     "T 127";
      =     "M 50.3";
NETWORK
TITLE =
      A     "M 50.3";
      CU    "Z 127";
      BLD   101;
      NOP   0;
      NOP   0;
      A     "M 59.3";
      R     "Z 127";
      NOP   0;
      LC    "Z 127";
      T     "MW 58";
      NOP   0;
NETWORK
TITLE =
      A     "M 59.0";
      =     "M 50.0";
NETWORK
TITLE =
      A     "M 59.1";
      =     "M 50.1";
NETWORK
TITLE =
      A     "M 59.2";
      =     "M 50.2";
END_FUNCTION

FUNCTION "FC 125" : VOID	// FC 125
VERSION : 0.1
BEGIN
// (block stored without names or comments; labels and parameter names are numbered)
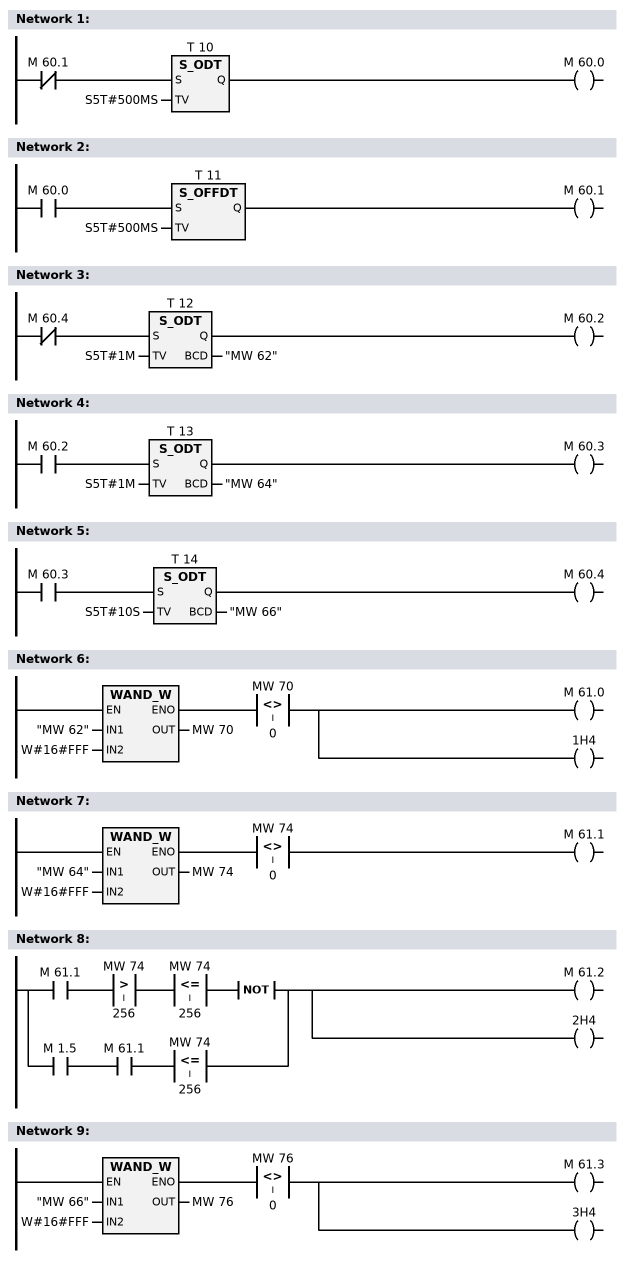
NETWORK
TITLE =
      AN    "M 60.1";
      L     S5T#500MS;
      SD    "T 10";
      NOP   0;
      NOP   0;
      NOP   0;
      A     "T 10";
      =     "M 60.0";
NETWORK
TITLE =
      A     "M 60.0";
      L     S5T#500MS;
      SF    "T 11";
      NOP   0;
      NOP   0;
      NOP   0;
      A     "T 11";
      =     "M 60.1";
NETWORK
TITLE =
      AN    "M 60.4";
      L     S5T#1M;
      SD    "T 12";
      NOP   0;
      NOP   0;
      LC    "T 12";
      T     "MW 62";
      A     "T 12";
      =     "M 60.2";
NETWORK
TITLE =
      A     "M 60.2";
      L     S5T#1M;
      SD    "T 13";
      NOP   0;
      NOP   0;
      LC    "T 13";
      T     "MW 64";
      A     "T 13";
      =     "M 60.3";
NETWORK
TITLE =
      A     "M 60.3";
      L     S5T#10S;
      SD    "T 14";
      NOP   0;
      NOP   0;
      LC    "T 14";
      T     "MW 66";
      A     "T 14";
      =     "M 60.4";
NETWORK
TITLE =
      A(;
      L     "MW 62";
      L     W#16#FFF;
      AW;
      T     MW 70;
      SET;
      SAVE;
      CLR;
      A     BR;
      );
      A(;
      L     MW 70;
      L     0;
      <>I;
      );
      =     "M 61.0";
      =     "1H4";
NETWORK
TITLE =
      A(;
      L     "MW 64";
      L     W#16#FFF;
      AW;
      T     MW 74;
      SET;
      SAVE;
      CLR;
      A     BR;
      );
      A(;
      L     MW 74;
      L     0;
      <>I;
      );
      =     "M 61.1";
NETWORK
TITLE =
      A     "M 61.1";
      A(;
      L     MW 74;
      L     256;
      >I;
      );
      A(;
      A(;
      L     MW 74;
      L     256;
      <=I;
      );
      NOT;
      );
      O;
      A     "M 1.5";
      A     "M 61.1";
      A(;
      L     MW 74;
      L     256;
      <=I;
      );
      =     "M 61.2";
      =     "2H4";
NETWORK
TITLE =
      A(;
      L     "MW 66";
      L     W#16#FFF;
      AW;
      T     MW 76;
      SET;
      SAVE;
      CLR;
      A     BR;
      );
      A(;
      L     MW 76;
      L     0;
      <>I;
      );
      =     "M 61.3";
      =     "3H4";
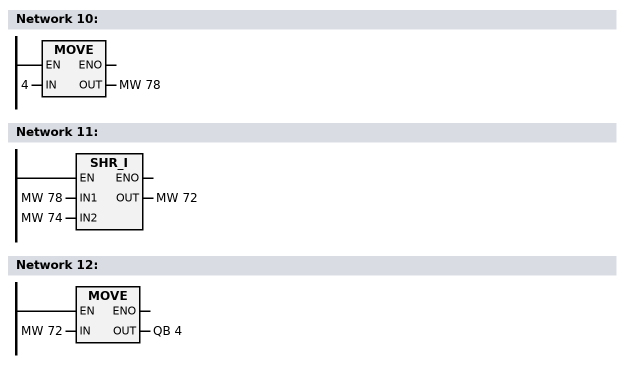
NETWORK
TITLE =
      L     4;
      T     MW 78;
      NOP   0;
NETWORK
TITLE =
      L     MW 78;
      L     MW 74;
      SSI;
      T     MW 72;
      NOP   0;
NETWORK
TITLE =
      L     MW 72;
      T     QB 4;
      NOP   0;
END_FUNCTION

FUNCTION "FC 130" : VOID	// FC 130
VERSION : 0.1
BEGIN
// (block stored without names or comments; labels and parameter names are numbered)
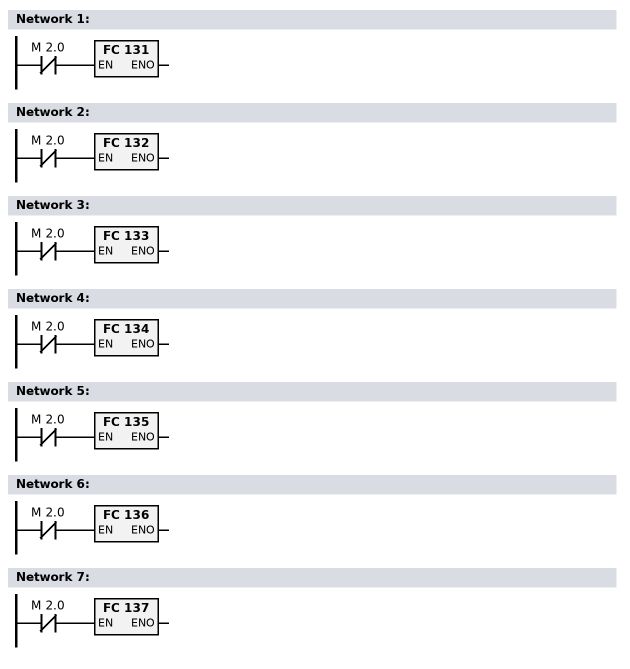
NETWORK
TITLE =
      AN    "M 2.0";
      JNB   M001;
      CALL  "FC 131";
M001: NOP   0;
NETWORK
TITLE =
      AN    "M 2.0";
      JNB   M002;
      CALL  "FC 132";
M002: NOP   0;
NETWORK
TITLE =
      AN    "M 2.0";
      JNB   M003;
      CALL  "FC 133";
M003: NOP   0;
NETWORK
TITLE =
      AN    "M 2.0";
      JNB   M004;
      CALL  "FC 134";
M004: NOP   0;
NETWORK
TITLE =
      AN    "M 2.0";
      JNB   M005;
      CALL  "FC 135";
M005: NOP   0;
NETWORK
TITLE =
      AN    "M 2.0";
      JNB   M006;
      CALL  "FC 136";
M006: NOP   0;
NETWORK
TITLE =
      AN    "M 2.0";
      JNB   M007;
      CALL  "FC 137";
M007: NOP   0;
END_FUNCTION

FUNCTION "FC 131" : VOID	// FC 131
VERSION : 0.1
BEGIN
// (block stored without names or comments; labels and parameter names are numbered)
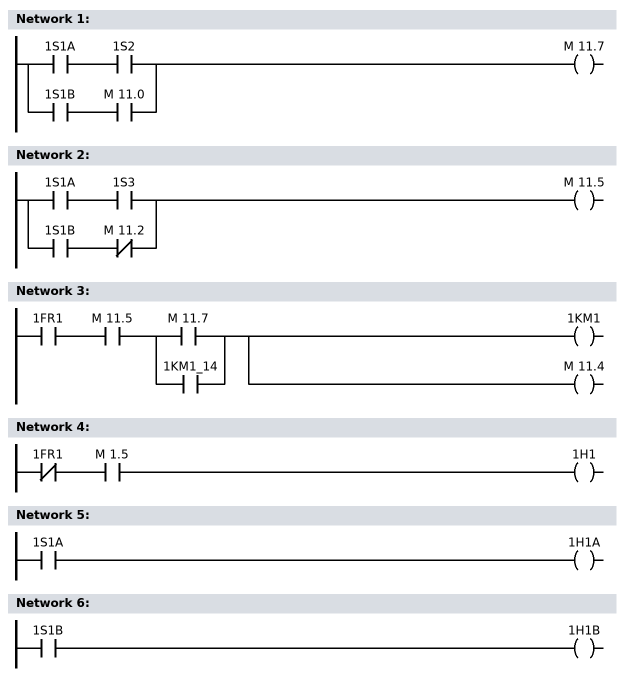
NETWORK
TITLE =
      A     "1S1A";
      A     "1S2";
      O;
      A     "1S1B";
      A     "M 11.0";
      =     "M 11.7";
NETWORK
TITLE =
      A     "1S1A";
      A     "1S3";
      O;
      A     "1S1B";
      AN    "M 11.2";
      =     "M 11.5";
NETWORK
TITLE =
      A     "1FR1";
      A     "M 11.5";
      A(;
      O     "M 11.7";
      O     "1KM1_14";
      );
      =     "1KM1";
      =     "M 11.4";
NETWORK
TITLE =
      AN    "1FR1";
      A     "M 1.5";
      =     "1H1";
NETWORK
TITLE =
      A     "1S1A";
      =     "1H1A";
NETWORK
TITLE =
      A     "1S1B";
      =     "1H1B";
END_FUNCTION

FUNCTION "FC 132" : VOID	// FC 132
VERSION : 0.1
BEGIN
// (block stored without names or comments; labels and parameter names are numbered)
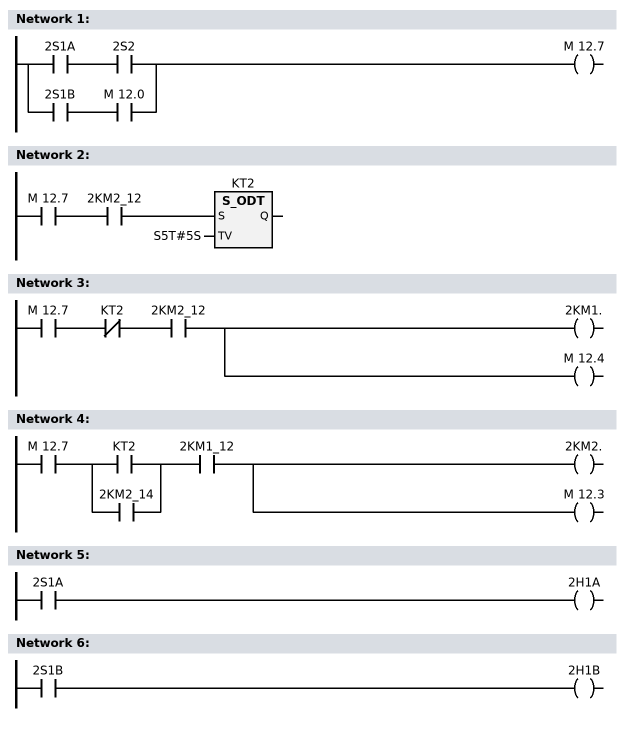
NETWORK
TITLE =
      A     "2S1A";
      A     "2S2";
      O;
      A     "2S1B";
      A     "M 12.0";
      =     "M 12.7";
NETWORK
TITLE =
      A     "M 12.7";
      A     "2KM2_12";
      L     S5T#5S;
      SD    "KT2";
      NOP   0;
      NOP   0;
      NOP   0;
      NOP   0;
NETWORK
TITLE =
      A     "M 12.7";
      AN    "KT2";
      A     "2KM2_12";
      =     "2KM1.";
      =     "M 12.4";
NETWORK
TITLE =
      A     "M 12.7";
      A(;
      O     "KT2";
      O     "2KM2_14";
      );
      A     "2KM1_12";
      =     "2KM2.";
      =     "M 12.3";
NETWORK
TITLE =
      A     "2S1A";
      =     "2H1A";
NETWORK
TITLE =
      A     "2S1B";
      =     "2H1B";
END_FUNCTION

FUNCTION "FC 133" : VOID	// FC 133
VERSION : 0.1
BEGIN
// (block stored without names or comments; labels and parameter names are numbered)
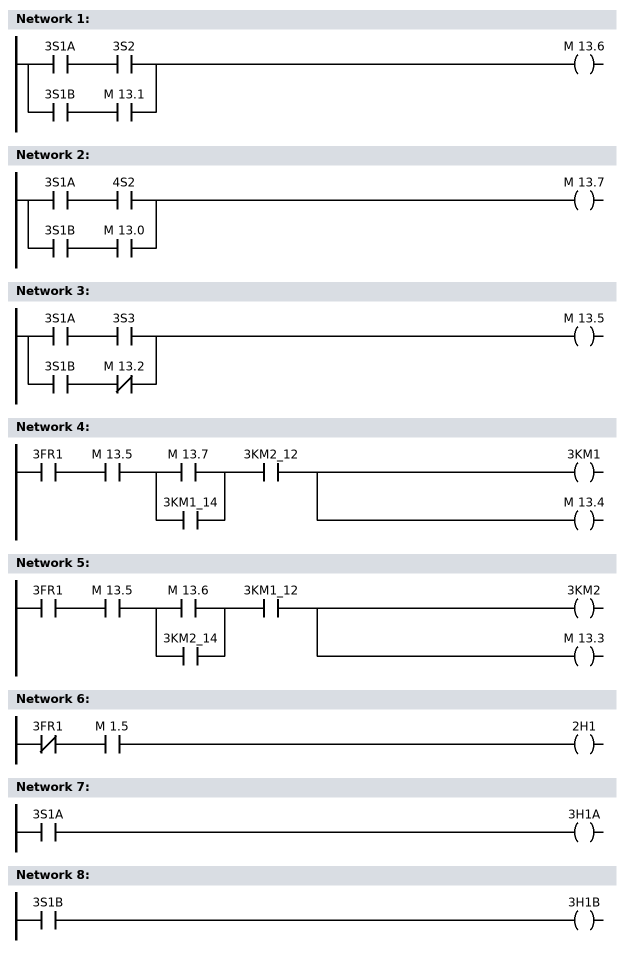
NETWORK
TITLE =
      A     "3S1A";
      A     "3S2";
      O;
      A     "3S1B";
      A     "M 13.1";
      =     "M 13.6";
NETWORK
TITLE =
      A     "3S1A";
      A     "4S2";
      O;
      A     "3S1B";
      A     "M 13.0";
      =     "M 13.7";
NETWORK
TITLE =
      A     "3S1A";
      A     "3S3";
      O;
      A     "3S1B";
      AN    "M 13.2";
      =     "M 13.5";
NETWORK
TITLE =
      A     "3FR1";
      A     "M 13.5";
      A(;
      O     "M 13.7";
      O     "3KM1_14";
      );
      A     "3KM2_12";
      =     "3KM1";
      =     "M 13.4";
NETWORK
TITLE =
      A     "3FR1";
      A     "M 13.5";
      A(;
      O     "M 13.6";
      O     "3KM2_14";
      );
      A     "3KM1_12";
      =     "3KM2";
      =     "M 13.3";
NETWORK
TITLE =
      AN    "3FR1";
      A     "M 1.5";
      =     "2H1";
NETWORK
TITLE =
      A     "3S1A";
      =     "3H1A";
NETWORK
TITLE =
      A     "3S1B";
      =     "3H1B";
END_FUNCTION

FUNCTION "FC 134" : VOID	// FC 134
VERSION : 0.1
BEGIN
// (block stored without names or comments; labels and parameter names are numbered)
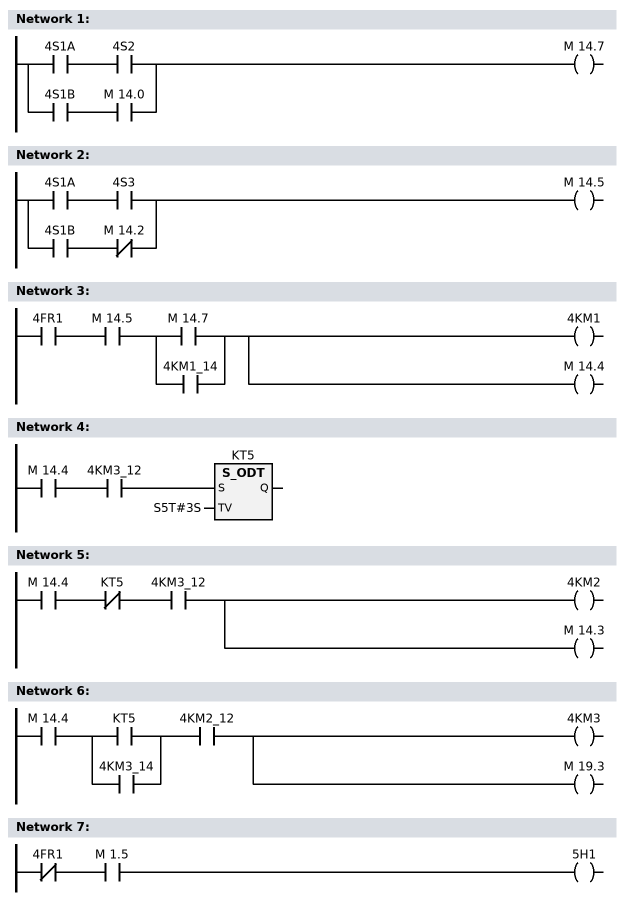
NETWORK
TITLE =
      A     "4S1A";
      A     "4S2";
      O;
      A     "4S1B";
      A     "M 14.0";
      =     "M 14.7";
NETWORK
TITLE =
      A     "4S1A";
      A     "4S3";
      O;
      A     "4S1B";
      AN    "M 14.2";
      =     "M 14.5";
NETWORK
TITLE =
      A     "4FR1";
      A     "M 14.5";
      A(;
      O     "M 14.7";
      O     "4KM1_14";
      );
      =     "4KM1";
      =     "M 14.4";
NETWORK
TITLE =
      A     "M 14.4";
      A     "4KM3_12";
      L     S5T#3S;
      SD    "KT5";
      NOP   0;
      NOP   0;
      NOP   0;
      NOP   0;
NETWORK
TITLE =
      A     "M 14.4";
      AN    "KT5";
      A     "4KM3_12";
      =     "4KM2";
      =     "M 14.3";
NETWORK
TITLE =
      A     "M 14.4";
      A(;
      O     "KT5";
      O     "4KM3_14";
      );
      A     "4KM2_12";
      =     "4KM3";
      =     "M 19.3";
NETWORK
TITLE =
      AN    "4FR1";
      A     "M 1.5";
      =     "5H1";
END_FUNCTION

FUNCTION "FC 135" : VOID	// FC 135
VERSION : 0.1
BEGIN
// (block stored without names or comments; labels and parameter names are numbered)
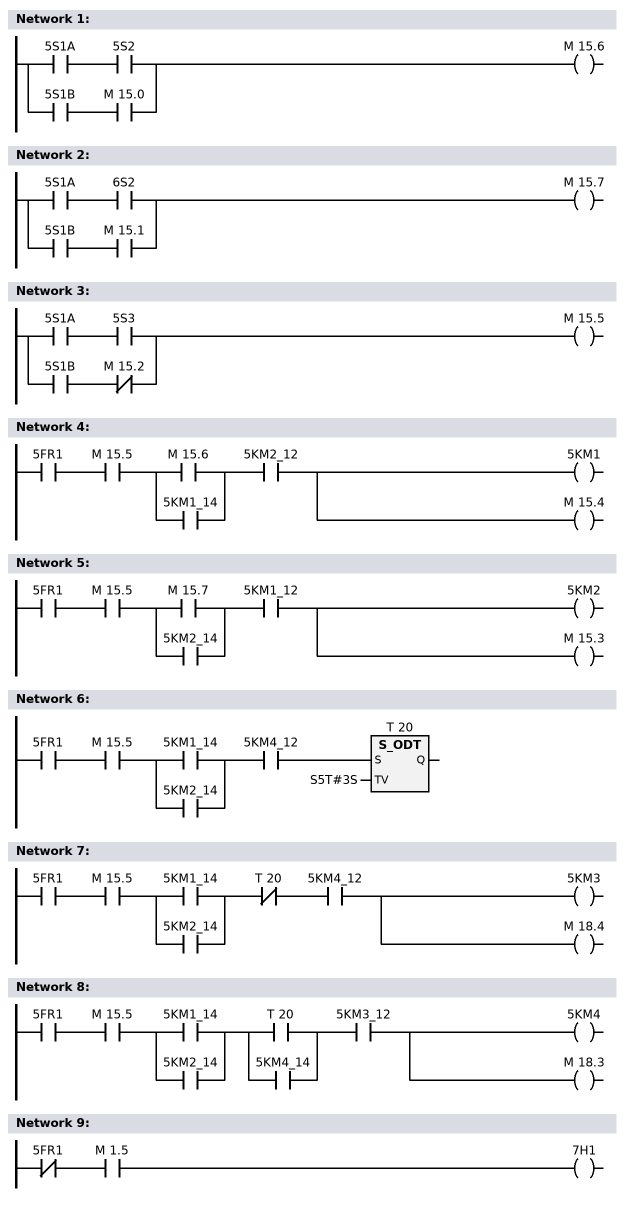
NETWORK
TITLE =
      A     "5S1A";
      A     "5S2";
      O;
      A     "5S1B";
      A     "M 15.0";
      =     "M 15.6";
NETWORK
TITLE =
      A     "5S1A";
      A     "6S2";
      O;
      A     "5S1B";
      A     "M 15.1";
      =     "M 15.7";
NETWORK
TITLE =
      A     "5S1A";
      A     "5S3";
      O;
      A     "5S1B";
      AN    "M 15.2";
      =     "M 15.5";
NETWORK
TITLE =
      A     "5FR1";
      A     "M 15.5";
      A(;
      O     "M 15.6";
      O     "5KM1_14";
      );
      A     "5KM2_12";
      =     "5KM1";
      =     "M 15.4";
NETWORK
TITLE =
      A     "5FR1";
      A     "M 15.5";
      A(;
      O     "M 15.7";
      O     "5KM2_14";
      );
      A     "5KM1_12";
      =     "5KM2";
      =     "M 15.3";
NETWORK
TITLE =
      A     "5FR1";
      A     "M 15.5";
      A(;
      O     "5KM1_14";
      O     "5KM2_14";
      );
      A     "5KM4_12";
      L     S5T#3S;
      SD    "T 20";
      NOP   0;
      NOP   0;
      NOP   0;
      NOP   0;
NETWORK
TITLE =
      A     "5FR1";
      A     "M 15.5";
      A(;
      O     "5KM1_14";
      O     "5KM2_14";
      );
      AN    "T 20";
      A     "5KM4_12";
      =     "5KM3";
      =     "M 18.4";
NETWORK
TITLE =
      A     "5FR1";
      A     "M 15.5";
      A(;
      O     "5KM1_14";
      O     "5KM2_14";
      );
      A(;
      O     "T 20";
      O     "5KM4_14";
      );
      A     "5KM3_12";
      =     "5KM4";
      =     "M 18.3";
NETWORK
TITLE =
      AN    "5FR1";
      A     "M 1.5";
      =     "7H1";
END_FUNCTION

FUNCTION "FC 136" : VOID	// FC 136
VERSION : 0.1
BEGIN
// (block stored without names or comments; labels and parameter names are numbered)
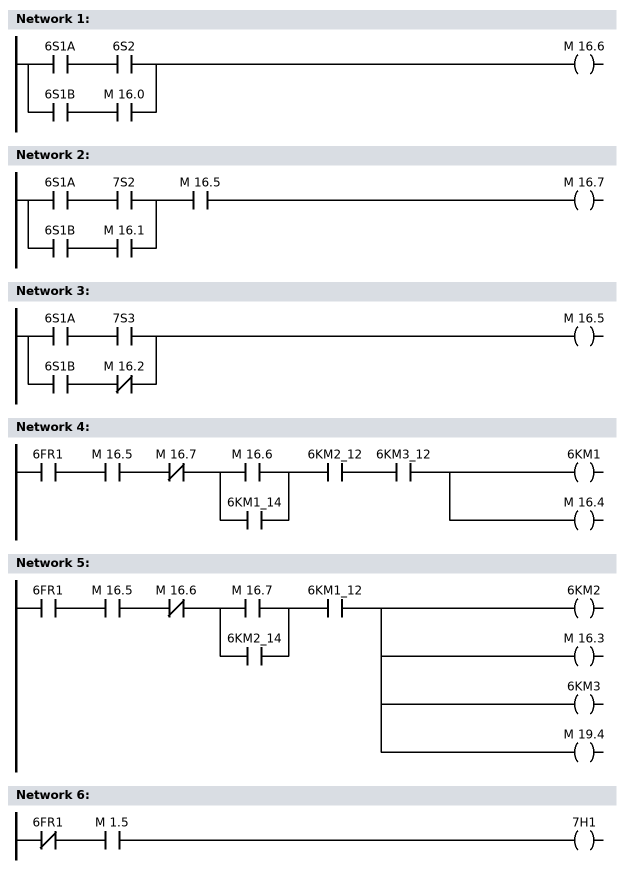
NETWORK
TITLE =
      A     "6S1A";
      A     "6S2";
      O;
      A     "6S1B";
      A     "M 16.0";
      =     "M 16.6";
NETWORK
TITLE =
      A(;
      A     "6S1A";
      A     "7S2";
      O;
      A     "6S1B";
      A     "M 16.1";
      );
      A     "M 16.5";
      =     "M 16.7";
NETWORK
TITLE =
      A     "6S1A";
      A     "7S3";
      O;
      A     "6S1B";
      AN    "M 16.2";
      =     "M 16.5";
NETWORK
TITLE =
      A     "6FR1";
      A     "M 16.5";
      AN    "M 16.7";
      A(;
      O     "M 16.6";
      O     "6KM1_14";
      );
      A     "6KM2_12";
      A     "6KM3_12";
      =     "6KM1";
      =     "M 16.4";
NETWORK
TITLE =
      A     "6FR1";
      A     "M 16.5";
      AN    "M 16.6";
      A(;
      O     "M 16.7";
      O     "6KM2_14";
      );
      A     "6KM1_12";
      =     "6KM2";
      =     "M 16.3";
      =     "6KM3";
      =     "M 19.4";
NETWORK
TITLE =
      AN    "6FR1";
      A     "M 1.5";
      =     "7H1";
END_FUNCTION

FUNCTION "FC 137" : VOID	// FC 137
VERSION : 0.1
BEGIN
// (block stored without names or comments; labels and parameter names are numbered)
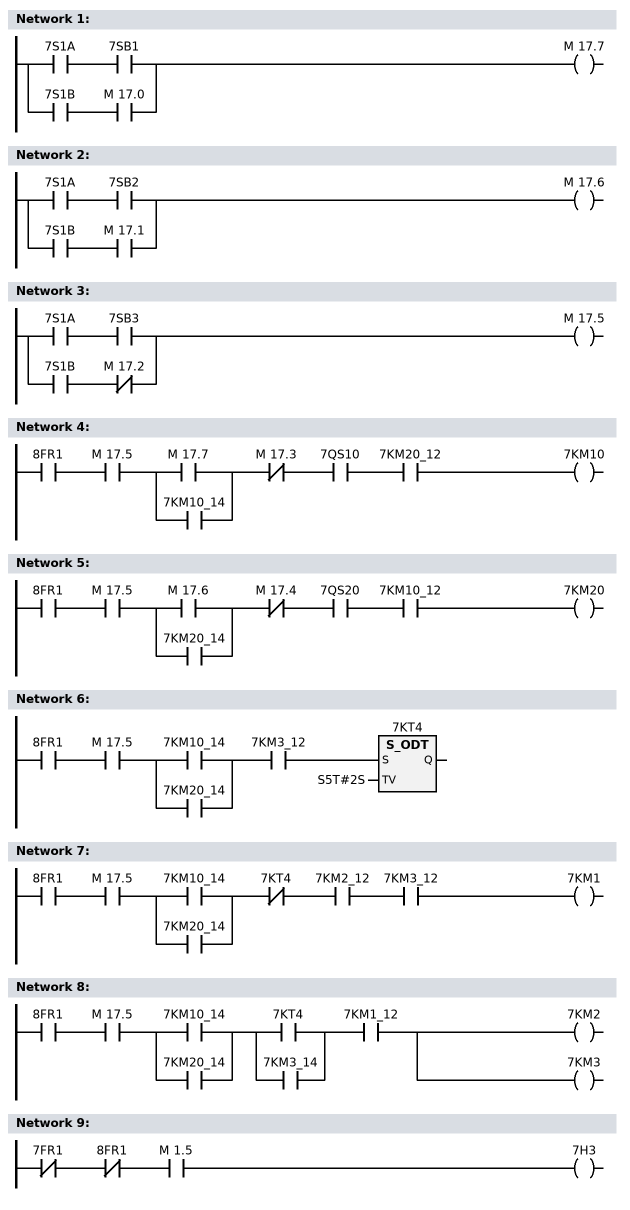
NETWORK
TITLE =
      A     "7S1A";
      A     "7SB1";
      O;
      A     "7S1B";
      A     "M 17.0";
      =     "M 17.7";
NETWORK
TITLE =
      A     "7S1A";
      A     "7SB2";
      O;
      A     "7S1B";
      A     "M 17.1";
      =     "M 17.6";
NETWORK
TITLE =
      A     "7S1A";
      A     "7SB3";
      O;
      A     "7S1B";
      AN    "M 17.2";
      =     "M 17.5";
NETWORK
TITLE =
      A     "8FR1";
      A     "M 17.5";
      A(;
      O     "M 17.7";
      O     "7KM10_14";
      );
      AN    "M 17.3";
      A     "7QS10";
      A     "7KM20_12";
      =     "7KM10";
NETWORK
TITLE =
      A     "8FR1";
      A     "M 17.5";
      A(;
      O     "M 17.6";
      O     "7KM20_14";
      );
      AN    "M 17.4";
      A     "7QS20";
      A     "7KM10_12";
      =     "7KM20";
NETWORK
TITLE =
      A     "8FR1";
      A     "M 17.5";
      A(;
      O     "7KM10_14";
      O     "7KM20_14";
      );
      A     "7KM3_12";
      L     S5T#2S;
      SD    "7KT4";
      NOP   0;
      NOP   0;
      NOP   0;
      NOP   0;
NETWORK
TITLE =
      A     "8FR1";
      A     "M 17.5";
      A(;
      O     "7KM10_14";
      O     "7KM20_14";
      );
      AN    "7KT4";
      A     "7KM2_12";
      A     "7KM3_12";
      =     "7KM1";
NETWORK
TITLE =
      A     "8FR1";
      A     "M 17.5";
      A(;
      O     "7KM10_14";
      O     "7KM20_14";
      );
      A(;
      O     "7KT4";
      O     "7KM3_14";
      );
      A     "7KM1_12";
      =     "7KM2";
      =     "7KM3";
NETWORK
TITLE =
      AN    "7FR1";
      AN    "8FR1";
      A     "M 1.5";
      =     "7H3";
END_FUNCTION

FUNCTION "FC 140" : VOID	// FC 140
VERSION : 0.1
BEGIN
// (block stored without names or comments; labels and parameter names are numbered)
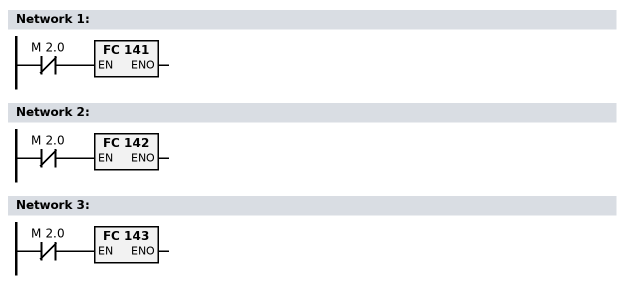
NETWORK
TITLE =
      AN    "M 2.0";
      JNB   M001;
      CALL  "FC 141";
M001: NOP   0;
NETWORK
TITLE =
      AN    "M 2.0";
      JNB   M002;
      CALL  "FC 142";
M002: NOP   0;
NETWORK
TITLE =
      AN    "M 2.0";
      JNB   M003;
      CALL  "FC 143";
M003: NOP   0;
END_FUNCTION

